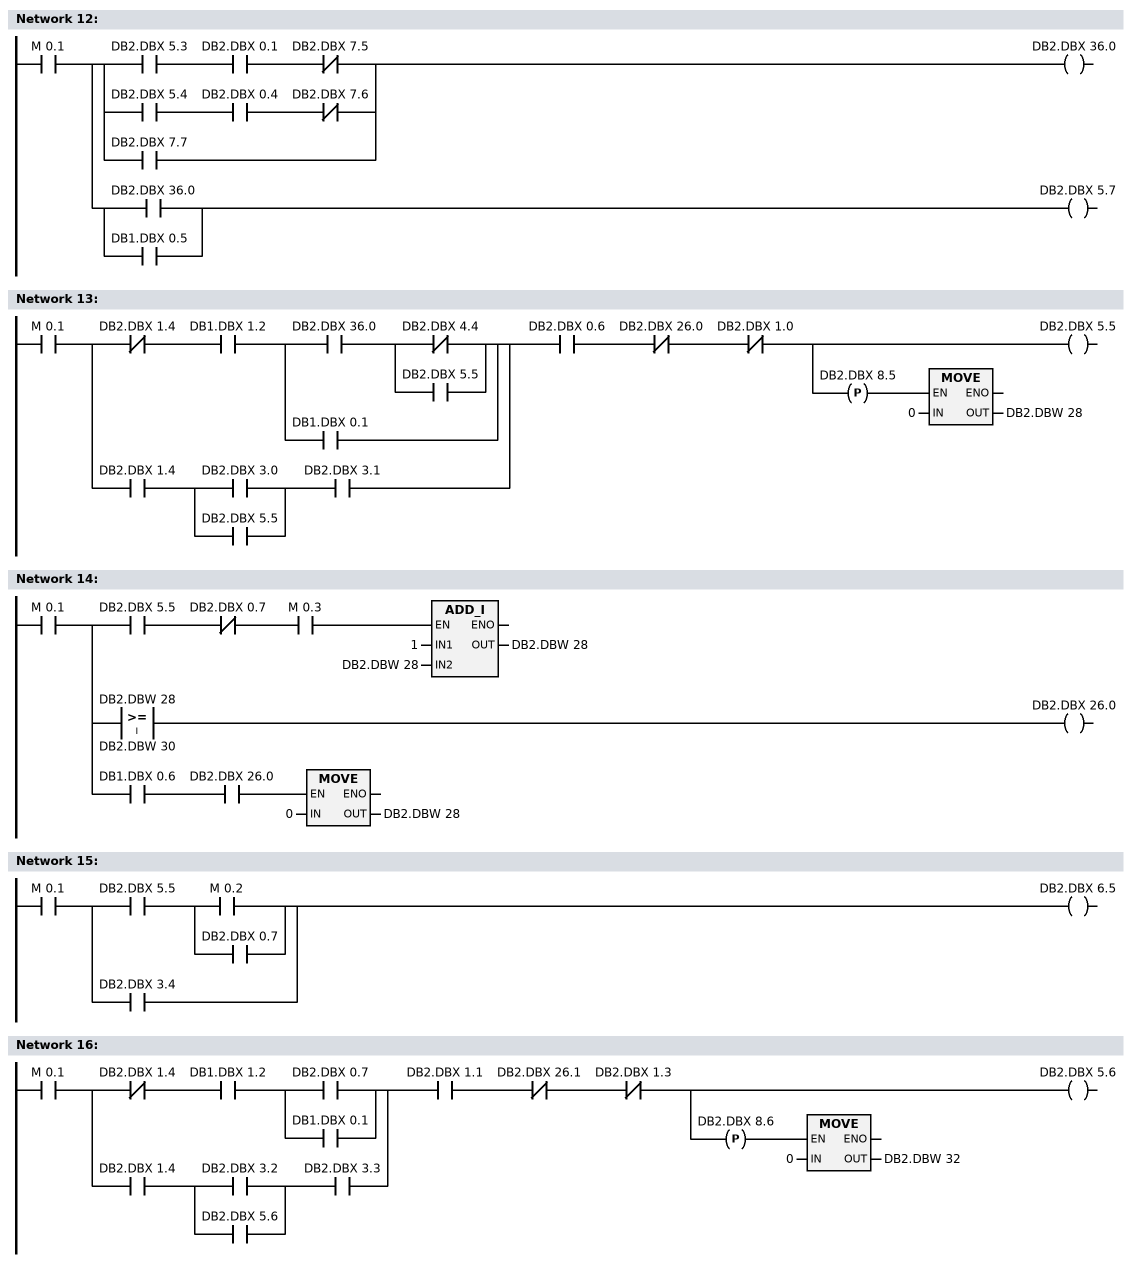
NETWORK
TITLE =
      A     M 0.1;
      =     L 0.0;
      A     L 0.0;
      A(;
      A     DB2.DBX 5.3;
      A     DB2.DBX 0.1;
      AN    DB2.DBX 7.5;
      O;
      A     DB2.DBX 5.4;
      A     DB2.DBX 0.4;
      AN    DB2.DBX 7.6;
      O     DB2.DBX 7.7;
      );
      =     DB2.DBX 36.0;
      A     L 0.0;
      A(;
      O     DB2.DBX 36.0;
      O     DB1.DBX 0.5;
      );
      =     DB2.DBX 5.7;
NETWORK
TITLE =
      A     M 0.1;
      A(;
      AN    DB2.DBX 1.4;
      A     DB1.DBX 1.2;
      A(;
      A     DB2.DBX 36.0;
      A(;
      ON    DB2.DBX 4.4;
      O     DB2.DBX 5.5;
      );
      O     DB1.DBX 0.1;
      );
      O;
      A     DB2.DBX 1.4;
      A(;
      O     DB2.DBX 3.0;
      O     DB2.DBX 5.5;
      );
      A     DB2.DBX 3.1;
      );
      A     DB2.DBX 0.6;
      AN    DB2.DBX 26.0;
      AN    DB2.DBX 1.0;
      =     L 0.0;
      A     L 0.0;
      BLD   102;
      =     DB2.DBX 5.5;
      A     L 0.0;
      FP    DB2.DBX 8.5;
      JNB   M011;
      L     0;
      T     DB2.DBW 28;
M011: NOP   0;
NETWORK
TITLE =
      A     M 0.1;
      =     L 0.0;
      A     L 0.0;
      A     DB2.DBX 5.5;
      AN    DB2.DBX 0.7;
      A     M 0.3;
      JNB   M012;
      L     1;
      L     DB2.DBW 28;
      +I;
      T     DB2.DBW 28;
M012: NOP   0;
      A     L 0.0;
      A(;
      L     DB2.DBW 28;
      L     DB2.DBW 30;
      >=I;
      );
      =     DB2.DBX 26.0;
      A     L 0.0;
      A     DB1.DBX 0.6;
      A     DB2.DBX 26.0;
      JNB   M013;
      L     0;
      T     DB2.DBW 28;
M013: NOP   0;
NETWORK
TITLE =
      A     M 0.1;
      A(;
      A     DB2.DBX 5.5;
      A(;
      O     M 0.2;
      O     DB2.DBX 0.7;
      );
      O     DB2.DBX 3.4;
      );
      =     DB2.DBX 6.5;
NETWORK
TITLE =
      A     M 0.1;
      A(;
      AN    DB2.DBX 1.4;
      A     DB1.DBX 1.2;
      A(;
      O     DB2.DBX 0.7;
      O     DB1.DBX 0.1;
      );
      O;
      A     DB2.DBX 1.4;
      A(;
      O     DB2.DBX 3.2;
      O     DB2.DBX 5.6;
      );
      A     DB2.DBX 3.3;
      );
      A     DB2.DBX 1.1;
      AN    DB2.DBX 26.1;
      AN    DB2.DBX 1.3;
      =     L 0.0;
      A     L 0.0;
      BLD   102;
      =     DB2.DBX 5.6;
      A     L 0.0;
      FP    DB2.DBX 8.6;
      JNB   M014;
      L     0;
      T     DB2.DBW 32;
M014: NOP   0;
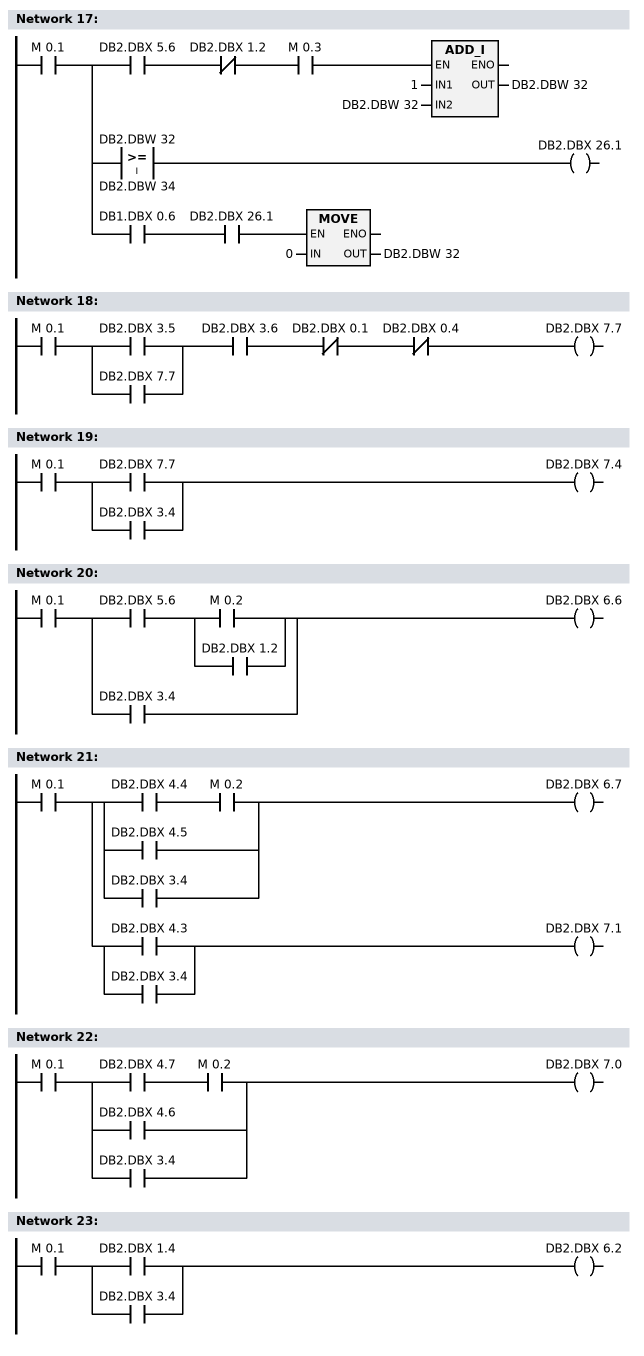
NETWORK
TITLE =
      A     M 0.1;
      =     L 0.0;
      A     L 0.0;
      A     DB2.DBX 5.6;
      AN    DB2.DBX 1.2;
      A     M 0.3;
      JNB   M015;
      L     1;
      L     DB2.DBW 32;
      +I;
      T     DB2.DBW 32;
M015: NOP   0;
      A     L 0.0;
      A(;
      L     DB2.DBW 32;
      L     DB2.DBW 34;
      >=I;
      );
      =     DB2.DBX 26.1;
      A     L 0.0;
      A     DB1.DBX 0.6;
      A     DB2.DBX 26.1;
      JNB   M016;
      L     0;
      T     DB2.DBW 32;
M016: NOP   0;
NETWORK
TITLE =
      A     M 0.1;
      A(;
      O     DB2.DBX 3.5;
      O     DB2.DBX 7.7;
      );
      A     DB2.DBX 3.6;
      AN    DB2.DBX 0.1;
      AN    DB2.DBX 0.4;
      =     DB2.DBX 7.7;
NETWORK
TITLE =
      A     M 0.1;
      A(;
      O     DB2.DBX 7.7;
      O     DB2.DBX 3.4;
      );
      =     DB2.DBX 7.4;
NETWORK
TITLE =
      A     M 0.1;
      A(;
      A     DB2.DBX 5.6;
      A(;
      O     M 0.2;
      O     DB2.DBX 1.2;
      );
      O     DB2.DBX 3.4;
      );
      =     DB2.DBX 6.6;
NETWORK
TITLE =
      A     M 0.1;
      =     L 0.0;
      A     L 0.0;
      A(;
      A     DB2.DBX 4.4;
      A     M 0.2;
      O     DB2.DBX 4.5;
      O     DB2.DBX 3.4;
      );
      =     DB2.DBX 6.7;
      A     L 0.0;
      A(;
      O     DB2.DBX 4.3;
      O     DB2.DBX 3.4;
      );
      =     DB2.DBX 7.1;
NETWORK
TITLE =
      A     M 0.1;
      A(;
      A     DB2.DBX 4.7;
      A     M 0.2;
      O     DB2.DBX 4.6;
      O     DB2.DBX 3.4;
      );
      =     DB2.DBX 7.0;
NETWORK
TITLE =
      A     M 0.1;
      A(;
      O     DB2.DBX 1.4;
      O     DB2.DBX 3.4;
      );
      =     DB2.DBX 6.2;
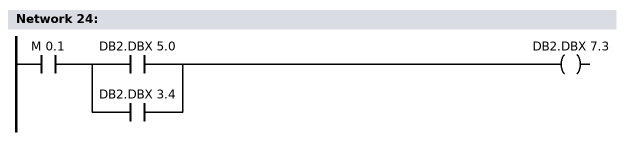
NETWORK
TITLE =
      A     M 0.1;
      A(;
      O     DB2.DBX 5.0;
      O     DB2.DBX 3.4;
      );
      =     DB2.DBX 7.3;
END_FUNCTION

FUNCTION FC 5 : VOID
AUTHOR : Kamillas
VERSION : 0.1
BEGIN
// (block stored without names or comments; labels and parameter names are numbered)
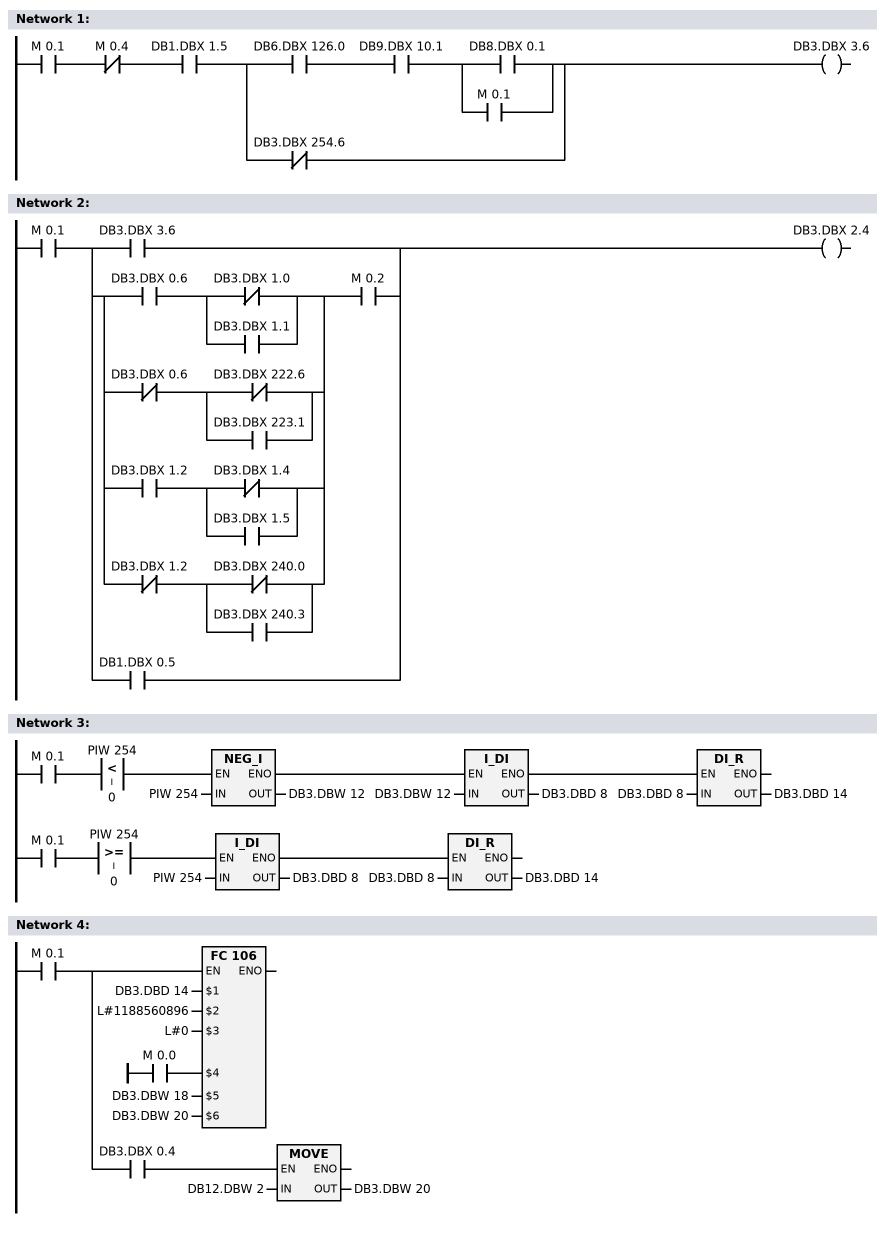
NETWORK
TITLE =
      A     M 0.1;
      AN    M 0.4;
      A     DB1.DBX 1.5;
      A(;
      A     DB6.DBX 126.0;
      A     DB9.DBX 10.1;
      A(;
      O     DB8.DBX 0.1;
      O     M 0.1;
      );
      ON    DB3.DBX 254.6;
      );
      =     DB3.DBX 3.6;
NETWORK
TITLE =
      A     M 0.1;
      A(;
      O     DB3.DBX 3.6;
      O;
      A(;
      A     DB3.DBX 0.6;
      A(;
      ON    DB3.DBX 1.0;
      O     DB3.DBX 1.1;
      );
      O;
      AN    DB3.DBX 0.6;
      A(;
      ON    DB3.DBX 222.6;
      O     DB3.DBX 223.1;
      );
      O;
      A     DB3.DBX 1.2;
      A(;
      ON    DB3.DBX 1.4;
      O     DB3.DBX 1.5;
      );
      O;
      AN    DB3.DBX 1.2;
      A(;
      ON    DB3.DBX 240.0;
      O     DB3.DBX 240.3;
      );
      );
      A     M 0.2;
      O     DB1.DBX 0.5;
      );
      =     DB3.DBX 2.4;
NETWORK
TITLE =
      A     M 0.1;
      =     L 0.0;
      A(;
      A(;
      A     L 0.0;
      A(;
      L     PIW 254;
      L     0;
      <I;
      );
      JNB   M001;
      L     PIW 254;
      NEGI;
      T     DB3.DBW 12;
      AN    OV;
      SAVE;
      CLR;
M001: A     BR;
      );
      JNB   M002;
      L     DB3.DBW 12;
      ITD;
      T     DB3.DBD 8;
      SET;
      SAVE;
      CLR;
M002: A     BR;
      );
      JNB   M003;
      L     DB3.DBD 8;
      DTR;
      T     DB3.DBD 14;
M003: NOP   0;
      A(;
      A     L 0.0;
      A(;
      L     PIW 254;
      L     0;
      >=I;
      );
      JNB   M004;
      L     PIW 254;
      ITD;
      T     DB3.DBD 8;
      SET;
      SAVE;
      CLR;
M004: A     BR;
      );
      JNB   M005;
      L     DB3.DBD 8;
      DTR;
      T     DB3.DBD 14;
M005: NOP   0;
NETWORK
TITLE =
      A     M 0.1;
      =     L 0.0;
      A     M 0.0;
      =     L 0.1;
      BLD   103;
      A     L 0.0;
      JNB   M006;
      CALL  FC 106 (
           $1                       := DB3.DBD 14,
           $2                       := L#1188560896,
           $3                       := L#0,
           $4                       := L 0.1,
           $5                       := DB3.DBW 18,
           $6                       := DB3.DBW 20);
M006: NOP   0;
      A     L 0.0;
      A     DB3.DBX 0.4;
      JNB   M007;
      L     DB12.DBW 2;
      T     DB3.DBW 20;
M007: NOP   0;
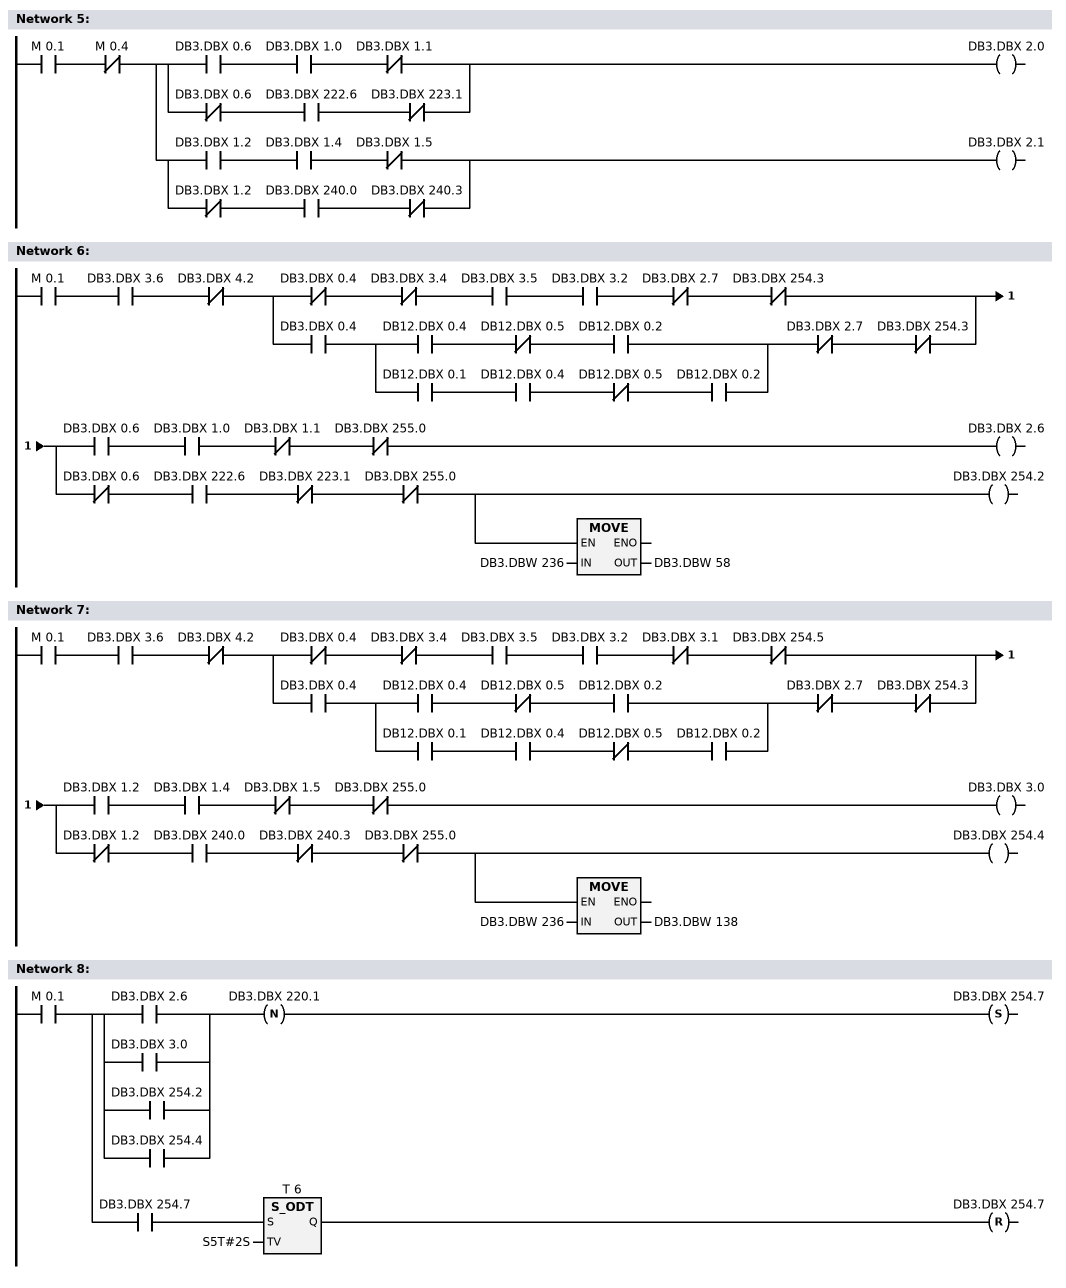
NETWORK
TITLE =
      A     M 0.1;
      AN    M 0.4;
      =     L 0.0;
      A     L 0.0;
      A(;
      A     DB3.DBX 0.6;
      A     DB3.DBX 1.0;
      AN    DB3.DBX 1.1;
      O;
      AN    DB3.DBX 0.6;
      A     DB3.DBX 222.6;
      AN    DB3.DBX 223.1;
      );
      =     DB3.DBX 2.0;
      A     L 0.0;
      A(;
      A     DB3.DBX 1.2;
      A     DB3.DBX 1.4;
      AN    DB3.DBX 1.5;
      O;
      AN    DB3.DBX 1.2;
      A     DB3.DBX 240.0;
      AN    DB3.DBX 240.3;
      );
      =     DB3.DBX 2.1;
NETWORK
TITLE =
      A     M 0.1;
      A     DB3.DBX 3.6;
      AN    DB3.DBX 4.2;
      A(;
      AN    DB3.DBX 0.4;
      AN    DB3.DBX 3.4;
      A     DB3.DBX 3.5;
      A     DB3.DBX 3.2;
      AN    DB3.DBX 2.7;
      AN    DB3.DBX 254.3;
      O;
      A     DB3.DBX 0.4;
      A(;
      A     DB12.DBX 0.4;
      AN    DB12.DBX 0.5;
      A     DB12.DBX 0.2;
      O;
      A     DB12.DBX 0.1;
      A     DB12.DBX 0.4;
      AN    DB12.DBX 0.5;
      A     DB12.DBX 0.2;
      );
      AN    DB3.DBX 2.7;
      AN    DB3.DBX 254.3;
      );
      =     L 0.0;
      A     L 0.0;
      A     DB3.DBX 0.6;
      A     DB3.DBX 1.0;
      AN    DB3.DBX 1.1;
      AN    DB3.DBX 255.0;
      =     DB3.DBX 2.6;
      A     L 0.0;
      AN    DB3.DBX 0.6;
      A     DB3.DBX 222.6;
      AN    DB3.DBX 223.1;
      AN    DB3.DBX 255.0;
      =     L 0.1;
      A     L 0.1;
      BLD   102;
      =     DB3.DBX 254.2;
      A     L 0.1;
      JNB   M008;
      L     DB3.DBW 236;
      T     DB3.DBW 58;
M008: NOP   0;
NETWORK
TITLE =
      A     M 0.1;
      A     DB3.DBX 3.6;
      AN    DB3.DBX 4.2;
      A(;
      AN    DB3.DBX 0.4;
      AN    DB3.DBX 3.4;
      A     DB3.DBX 3.5;
      A     DB3.DBX 3.2;
      AN    DB3.DBX 3.1;
      AN    DB3.DBX 254.5;
      O;
      A     DB3.DBX 0.4;
      A(;
      A     DB12.DBX 0.4;
      AN    DB12.DBX 0.5;
      A     DB12.DBX 0.2;
      O;
      A     DB12.DBX 0.1;
      A     DB12.DBX 0.4;
      AN    DB12.DBX 0.5;
      A     DB12.DBX 0.2;
      );
      AN    DB3.DBX 2.7;
      AN    DB3.DBX 254.3;
      );
      =     L 0.0;
      A     L 0.0;
      A     DB3.DBX 1.2;
      A     DB3.DBX 1.4;
      AN    DB3.DBX 1.5;
      AN    DB3.DBX 255.0;
      =     DB3.DBX 3.0;
      A     L 0.0;
      AN    DB3.DBX 1.2;
      A     DB3.DBX 240.0;
      AN    DB3.DBX 240.3;
      AN    DB3.DBX 255.0;
      =     L 0.1;
      A     L 0.1;
      BLD   102;
      =     DB3.DBX 254.4;
      A     L 0.1;
      JNB   M009;
      L     DB3.DBW 236;
      T     DB3.DBW 138;
M009: NOP   0;
NETWORK
TITLE =
      A     M 0.1;
      =     L 0.0;
      A     L 0.0;
      A(;
      O     DB3.DBX 2.6;
      O     DB3.DBX 3.0;
      O     DB3.DBX 254.2;
      O     DB3.DBX 254.4;
      );
      FN    DB3.DBX 220.1;
      S     DB3.DBX 254.7;
      A     L 0.0;
      A     DB3.DBX 254.7;
      L     S5T#2S;
      SD    T 6;
      NOP   0;
      NOP   0;
      NOP   0;
      A     T 6;
      R     DB3.DBX 254.7;
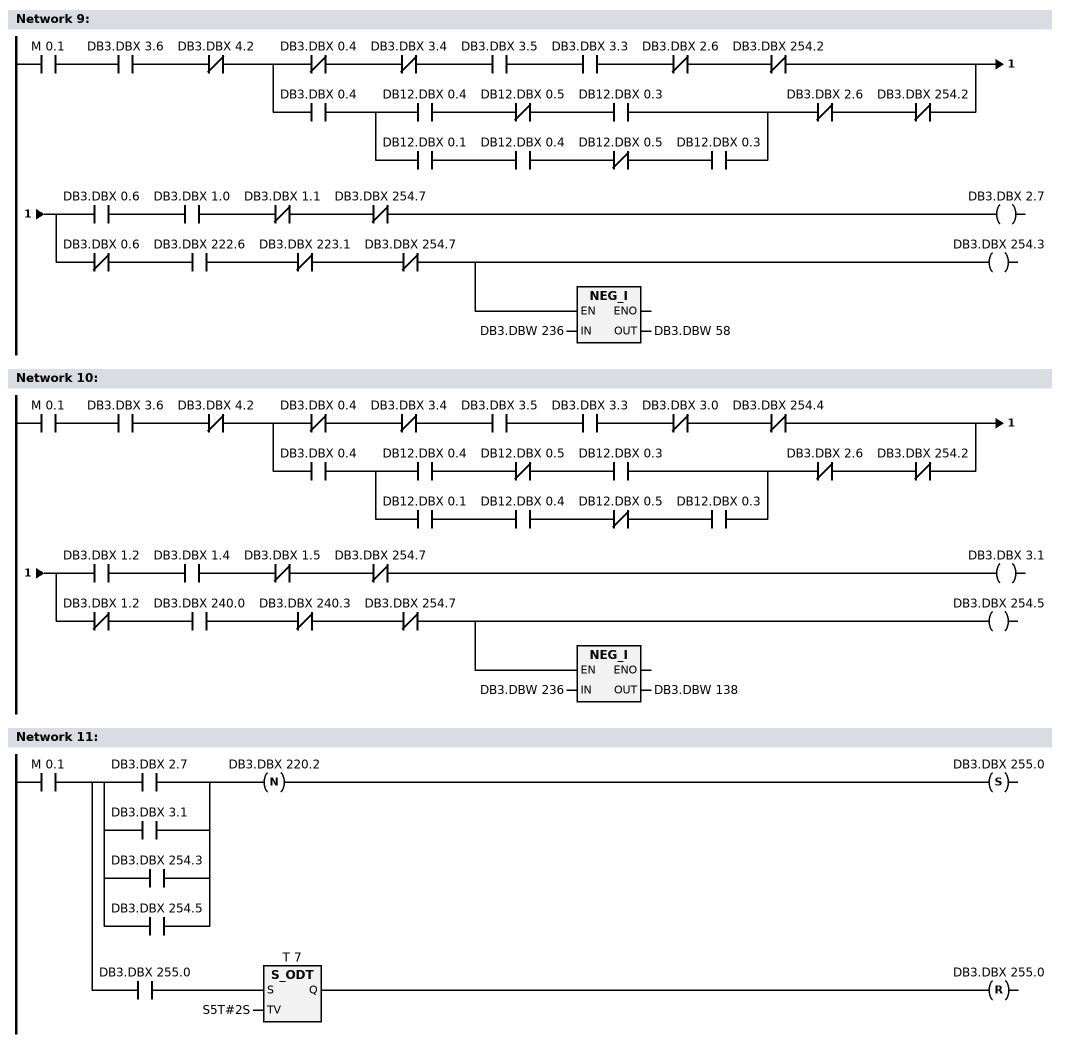
NETWORK
TITLE =
      A     M 0.1;
      A     DB3.DBX 3.6;
      AN    DB3.DBX 4.2;
      A(;
      AN    DB3.DBX 0.4;
      AN    DB3.DBX 3.4;
      A     DB3.DBX 3.5;
      A     DB3.DBX 3.3;
      AN    DB3.DBX 2.6;
      AN    DB3.DBX 254.2;
      O;
      A     DB3.DBX 0.4;
      A(;
      A     DB12.DBX 0.4;
      AN    DB12.DBX 0.5;
      A     DB12.DBX 0.3;
      O;
      A     DB12.DBX 0.1;
      A     DB12.DBX 0.4;
      AN    DB12.DBX 0.5;
      A     DB12.DBX 0.3;
      );
      AN    DB3.DBX 2.6;
      AN    DB3.DBX 254.2;
      );
      =     L 0.0;
      A     L 0.0;
      A     DB3.DBX 0.6;
      A     DB3.DBX 1.0;
      AN    DB3.DBX 1.1;
      AN    DB3.DBX 254.7;
      =     DB3.DBX 2.7;
      A     L 0.0;
      AN    DB3.DBX 0.6;
      A     DB3.DBX 222.6;
      AN    DB3.DBX 223.1;
      AN    DB3.DBX 254.7;
      =     L 0.1;
      A     L 0.1;
      BLD   102;
      =     DB3.DBX 254.3;
      A     L 0.1;
      JNB   M010;
      L     DB3.DBW 236;
      NEGI;
      T     DB3.DBW 58;
M010: NOP   0;
NETWORK
TITLE =
      A     M 0.1;
      A     DB3.DBX 3.6;
      AN    DB3.DBX 4.2;
      A(;
      AN    DB3.DBX 0.4;
      AN    DB3.DBX 3.4;
      A     DB3.DBX 3.5;
      A     DB3.DBX 3.3;
      AN    DB3.DBX 3.0;
      AN    DB3.DBX 254.4;
      O;
      A     DB3.DBX 0.4;
      A(;
      A     DB12.DBX 0.4;
      AN    DB12.DBX 0.5;
      A     DB12.DBX 0.3;
      O;
      A     DB12.DBX 0.1;
      A     DB12.DBX 0.4;
      AN    DB12.DBX 0.5;
      A     DB12.DBX 0.3;
      );
      AN    DB3.DBX 2.6;
      AN    DB3.DBX 254.2;
      );
      =     L 0.0;
      A     L 0.0;
      A     DB3.DBX 1.2;
      A     DB3.DBX 1.4;
      AN    DB3.DBX 1.5;
      AN    DB3.DBX 254.7;
      =     DB3.DBX 3.1;
      A     L 0.0;
      AN    DB3.DBX 1.2;
      A     DB3.DBX 240.0;
      AN    DB3.DBX 240.3;
      AN    DB3.DBX 254.7;
      =     L 0.1;
      A     L 0.1;
      BLD   102;
      =     DB3.DBX 254.5;
      A     L 0.1;
      JNB   M011;
      L     DB3.DBW 236;
      NEGI;
      T     DB3.DBW 138;
M011: NOP   0;
NETWORK
TITLE =
      A     M 0.1;
      =     L 0.0;
      A     L 0.0;
      A(;
      O     DB3.DBX 2.7;
      O     DB3.DBX 3.1;
      O     DB3.DBX 254.3;
      O     DB3.DBX 254.5;
      );
      FN    DB3.DBX 220.2;
      S     DB3.DBX 255.0;
      A     L 0.0;
      A     DB3.DBX 255.0;
      L     S5T#2S;
      SD    T 7;
      NOP   0;
      NOP   0;
      NOP   0;
      A     T 7;
      R     DB3.DBX 255.0;
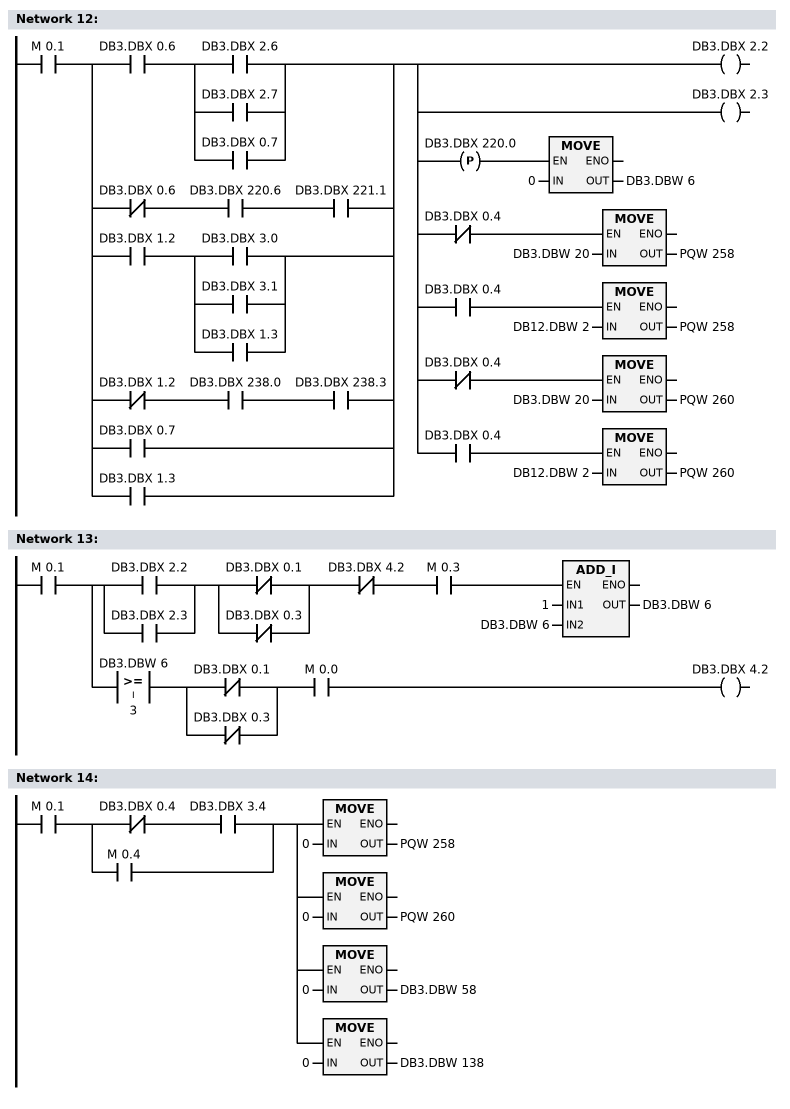
NETWORK
TITLE =
      A     M 0.1;
      A(;
      A     DB3.DBX 0.6;
      A(;
      O     DB3.DBX 2.6;
      O     DB3.DBX 2.7;
      O     DB3.DBX 0.7;
      );
      O;
      AN    DB3.DBX 0.6;
      A     DB3.DBX 220.6;
      A     DB3.DBX 221.1;
      O;
      A     DB3.DBX 1.2;
      A(;
      O     DB3.DBX 3.0;
      O     DB3.DBX 3.1;
      O     DB3.DBX 1.3;
      );
      O;
      AN    DB3.DBX 1.2;
      A     DB3.DBX 238.0;
      A     DB3.DBX 238.3;
      O     DB3.DBX 0.7;
      O     DB3.DBX 1.3;
      );
      =     L 0.0;
      A     L 0.0;
      BLD   102;
      =     DB3.DBX 2.2;
      A     L 0.0;
      BLD   102;
      =     DB3.DBX 2.3;
      A     L 0.0;
      FP    DB3.DBX 220.0;
      JNB   M012;
      L     0;
      T     DB3.DBW 6;
M012: NOP   0;
      A     L 0.0;
      AN    DB3.DBX 0.4;
      JNB   M013;
      L     DB3.DBW 20;
      T     PQW 258;
M013: NOP   0;
      A     L 0.0;
      A     DB3.DBX 0.4;
      JNB   M014;
      L     DB12.DBW 2;
      T     PQW 258;
M014: NOP   0;
      A     L 0.0;
      AN    DB3.DBX 0.4;
      JNB   M015;
      L     DB3.DBW 20;
      T     PQW 260;
M015: NOP   0;
      A     L 0.0;
      A     DB3.DBX 0.4;
      JNB   M016;
      L     DB12.DBW 2;
      T     PQW 260;
M016: NOP   0;
NETWORK
TITLE =
      A     M 0.1;
      =     L 0.0;
      A     L 0.0;
      A(;
      O     DB3.DBX 2.2;
      O     DB3.DBX 2.3;
      );
      A(;
      ON    DB3.DBX 0.1;
      ON    DB3.DBX 0.3;
      );
      AN    DB3.DBX 4.2;
      A     M 0.3;
      JNB   M017;
      L     1;
      L     DB3.DBW 6;
      +I;
      T     DB3.DBW 6;
M017: NOP   0;
      A     L 0.0;
      A(;
      L     DB3.DBW 6;
      L     3;
      >=I;
      );
      A(;
      ON    DB3.DBX 0.1;
      ON    DB3.DBX 0.3;
      );
      A     M 0.0;
      =     DB3.DBX 4.2;
NETWORK
TITLE =
      A     M 0.1;
      A(;
      AN    DB3.DBX 0.4;
      A     DB3.DBX 3.4;
      O     M 0.4;
      );
      =     L 0.0;
      A     L 0.0;
      JNB   M018;
      L     0;
      T     PQW 258;
M018: NOP   0;
      A     L 0.0;
      JNB   M019;
      L     0;
      T     PQW 260;
M019: NOP   0;
      A     L 0.0;
      JNB   M020;
      L     0;
      T     DB3.DBW 58;
M020: NOP   0;
      A     L 0.0;
      JNB   M021;
      L     0;
      T     DB3.DBW 138;
M021: NOP   0;
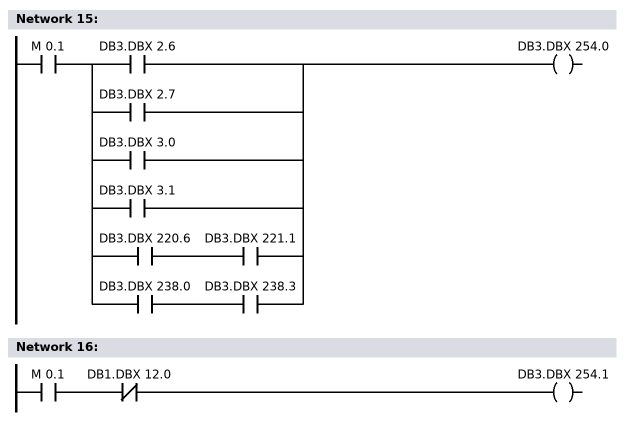
NETWORK
TITLE =
      A     M 0.1;
      A(;
      O     DB3.DBX 2.6;
      O     DB3.DBX 2.7;
      O     DB3.DBX 3.0;
      O     DB3.DBX 3.1;
      O;
      A     DB3.DBX 220.6;
      A     DB3.DBX 221.1;
      O;
      A     DB3.DBX 238.0;
      A     DB3.DBX 238.3;
      );
      =     DB3.DBX 254.0;
NETWORK
TITLE =
      A     M 0.1;
      AN    DB1.DBX 12.0;
      =     DB3.DBX 254.1;
END_FUNCTION

FUNCTION FC 6 : VOID
AUTHOR : Kamillas
VERSION : 0.1
BEGIN
// (block stored without names or comments; labels and parameter names are numbered)
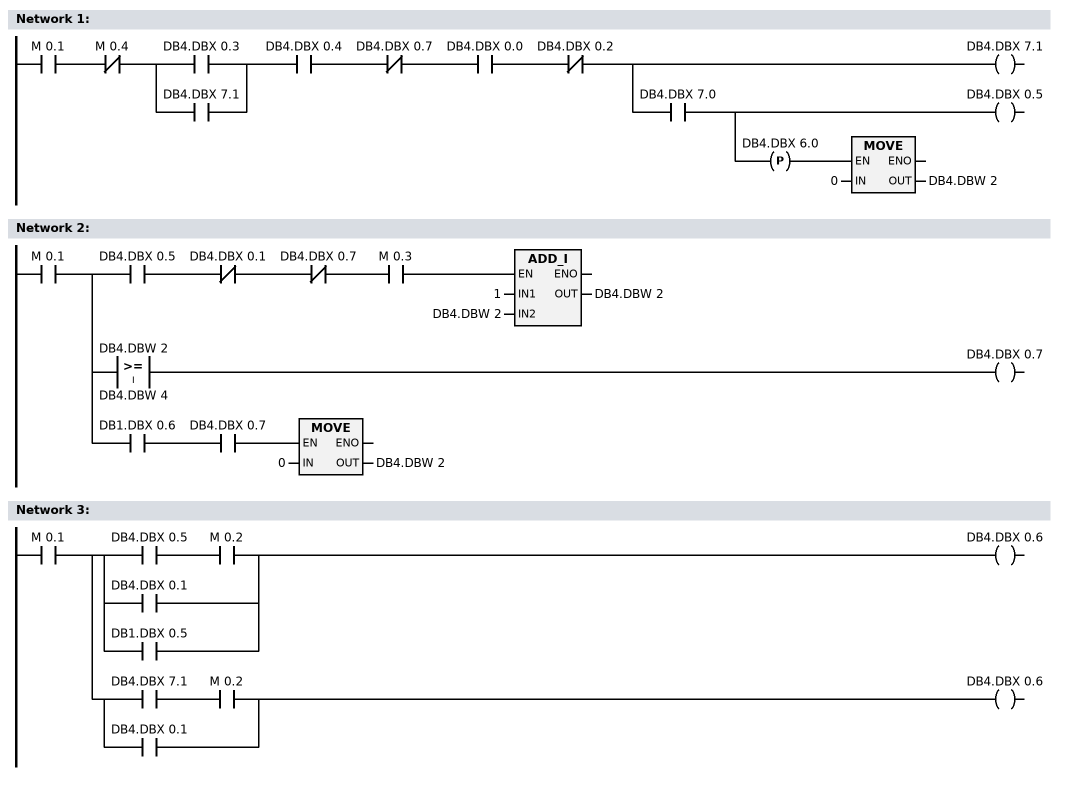
NETWORK
TITLE =
      A     M 0.1;
      AN    M 0.4;
      A(;
      O     DB4.DBX 0.3;
      O     DB4.DBX 7.1;
      );
      A     DB4.DBX 0.4;
      AN    DB4.DBX 0.7;
      A     DB4.DBX 0.0;
      AN    DB4.DBX 0.2;
      =     L 0.0;
      A     L 0.0;
      BLD   102;
      =     DB4.DBX 7.1;
      A     L 0.0;
      A     DB4.DBX 7.0;
      =     L 0.1;
      A     L 0.1;
      BLD   102;
      =     DB4.DBX 0.5;
      A     L 0.1;
      FP    DB4.DBX 6.0;
      JNB   M001;
      L     0;
      T     DB4.DBW 2;
M001: NOP   0;
NETWORK
TITLE =
      A     M 0.1;
      =     L 0.0;
      A     L 0.0;
      A     DB4.DBX 0.5;
      AN    DB4.DBX 0.1;
      AN    DB4.DBX 0.7;
      A     M 0.3;
      JNB   M002;
      L     1;
      L     DB4.DBW 2;
      +I;
      T     DB4.DBW 2;
M002: NOP   0;
      A     L 0.0;
      A(;
      L     DB4.DBW 2;
      L     DB4.DBW 4;
      >=I;
      );
      =     DB4.DBX 0.7;
      A     L 0.0;
      A     DB1.DBX 0.6;
      A     DB4.DBX 0.7;
      JNB   M003;
      L     0;
      T     DB4.DBW 2;
M003: NOP   0;
NETWORK
TITLE =
      A     M 0.1;
      =     L 0.0;
      A     L 0.0;
      A(;
      A     DB4.DBX 0.5;
      A     M 0.2;
      O     DB4.DBX 0.1;
      O     DB1.DBX 0.5;
      );
      =     DB4.DBX 0.6;
      A     L 0.0;
      A(;
      A     DB4.DBX 7.1;
      A     M 0.2;
      O     DB4.DBX 0.1;
      );
      =     DB4.DBX 0.6;
END_FUNCTION

FUNCTION FC 7 : VOID
AUTHOR : Kamillas
VERSION : 0.1
BEGIN
// (block stored without names or comments; labels and parameter names are numbered)
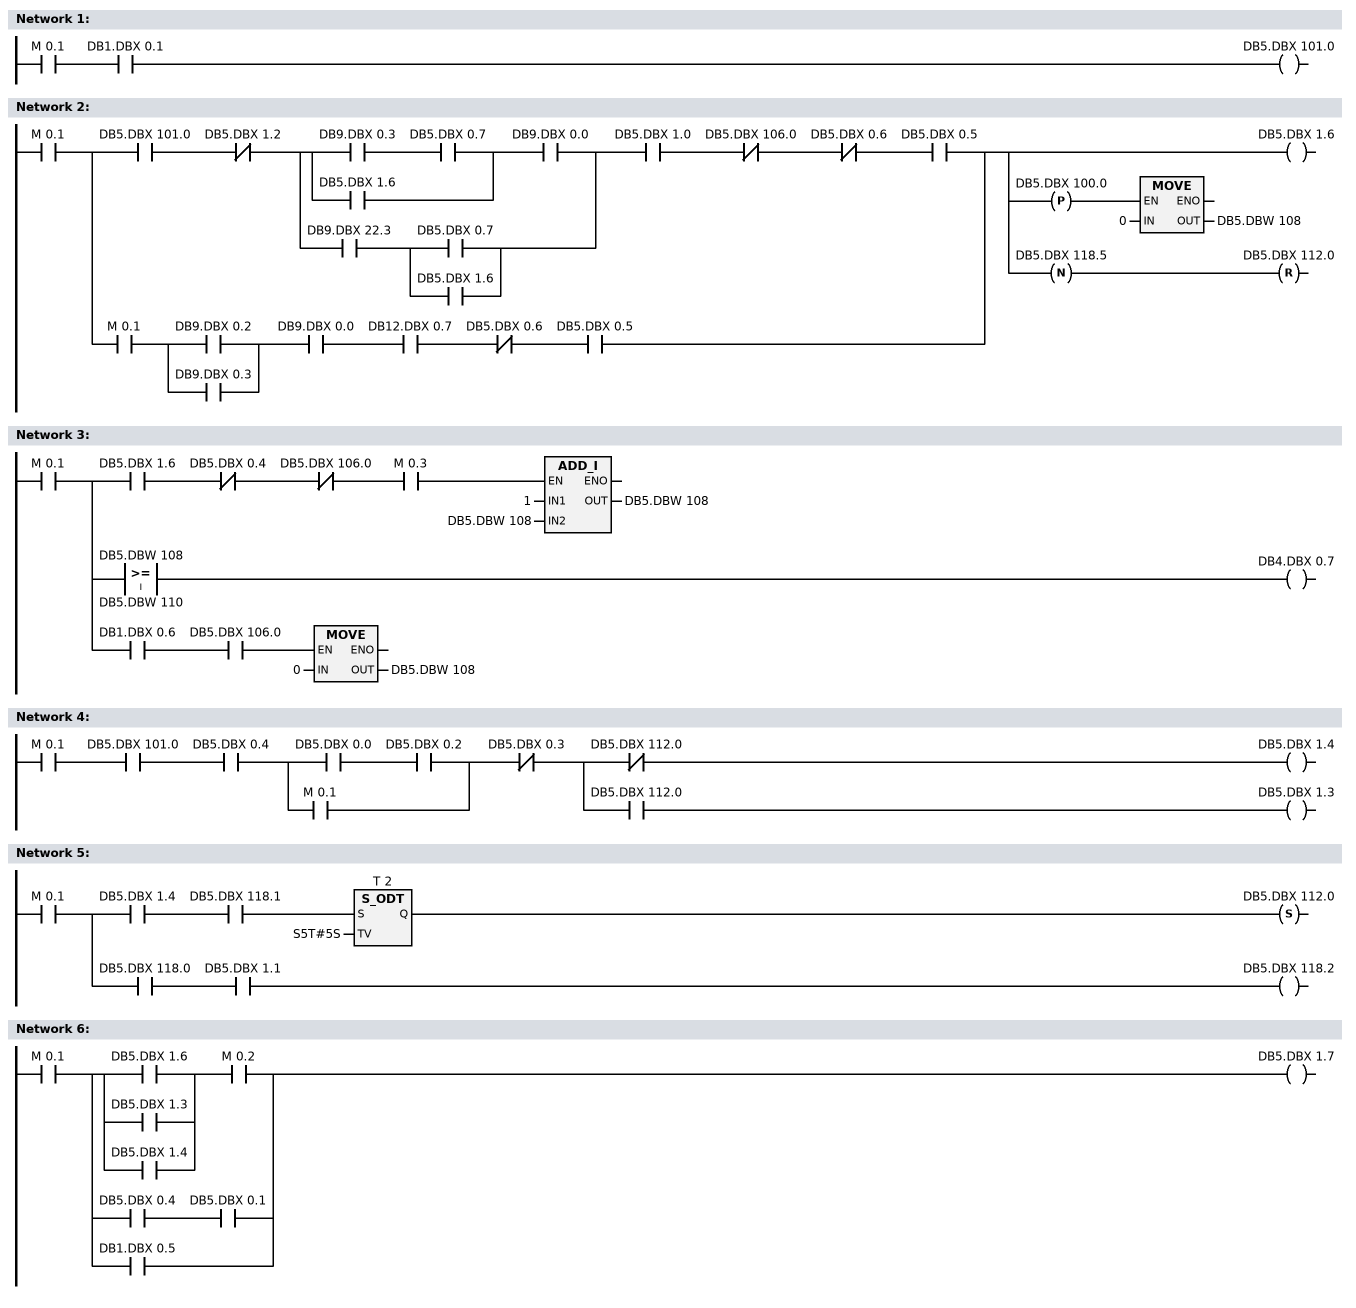
NETWORK
TITLE =
      A     M 0.1;
      A     DB1.DBX 0.1;
      =     DB5.DBX 101.0;
NETWORK
TITLE =
      A     M 0.1;
      A(;
      A     DB5.DBX 101.0;
      AN    DB5.DBX 1.2;
      A(;
      A(;
      A     DB9.DBX 0.3;
      A     DB5.DBX 0.7;
      O     DB5.DBX 1.6;
      );
      A     DB9.DBX 0.0;
      O;
      A     DB9.DBX 22.3;
      A(;
      O     DB5.DBX 0.7;
      O     DB5.DBX 1.6;
      );
      );
      A     DB5.DBX 1.0;
      AN    DB5.DBX 106.0;
      AN    DB5.DBX 0.6;
      A     DB5.DBX 0.5;
      O;
      A     M 0.1;
      A(;
      O     DB9.DBX 0.2;
      O     DB9.DBX 0.3;
      );
      A     DB9.DBX 0.0;
      A     DB12.DBX 0.7;
      AN    DB5.DBX 0.6;
      A     DB5.DBX 0.5;
      );
      =     L 0.0;
      A     L 0.0;
      BLD   102;
      =     DB5.DBX 1.6;
      A     L 0.0;
      FP    DB5.DBX 100.0;
      JNB   M001;
      L     0;
      T     DB5.DBW 108;
M001: NOP   0;
      A     L 0.0;
      FN    DB5.DBX 118.5;
      R     DB5.DBX 112.0;
NETWORK
TITLE =
      A     M 0.1;
      =     L 0.0;
      A     L 0.0;
      A     DB5.DBX 1.6;
      AN    DB5.DBX 0.4;
      AN    DB5.DBX 106.0;
      A     M 0.3;
      JNB   M002;
      L     1;
      L     DB5.DBW 108;
      +I;
      T     DB5.DBW 108;
M002: NOP   0;
      A     L 0.0;
      A(;
      L     DB5.DBW 108;
      L     DB5.DBW 110;
      >=I;
      );
      =     DB4.DBX 0.7;
      A     L 0.0;
      A     DB1.DBX 0.6;
      A     DB5.DBX 106.0;
      JNB   M003;
      L     0;
      T     DB5.DBW 108;
M003: NOP   0;
NETWORK
TITLE =
      A     M 0.1;
      A     DB5.DBX 101.0;
      A     DB5.DBX 0.4;
      A(;
      A     DB5.DBX 0.0;
      A     DB5.DBX 0.2;
      O     M 0.1;
      );
      AN    DB5.DBX 0.3;
      =     L 0.0;
      A     L 0.0;
      AN    DB5.DBX 112.0;
      =     DB5.DBX 1.4;
      A     L 0.0;
      A     DB5.DBX 112.0;
      =     DB5.DBX 1.3;
NETWORK
TITLE =
      A     M 0.1;
      =     L 0.0;
      A     L 0.0;
      A     DB5.DBX 1.4;
      A     DB5.DBX 118.1;
      L     S5T#5S;
      SD    T 2;
      NOP   0;
      NOP   0;
      NOP   0;
      A     T 2;
      S     DB5.DBX 112.0;
      A     L 0.0;
      A     DB5.DBX 118.0;
      A     DB5.DBX 1.1;
      =     DB5.DBX 118.2;
NETWORK
TITLE =
      A     M 0.1;
      A(;
      A(;
      O     DB5.DBX 1.6;
      O     DB5.DBX 1.3;
      O     DB5.DBX 1.4;
      );
      A     M 0.2;
      O;
      A     DB5.DBX 0.4;
      A     DB5.DBX 0.1;
      O     DB1.DBX 0.5;
      );
      =     DB5.DBX 1.7;
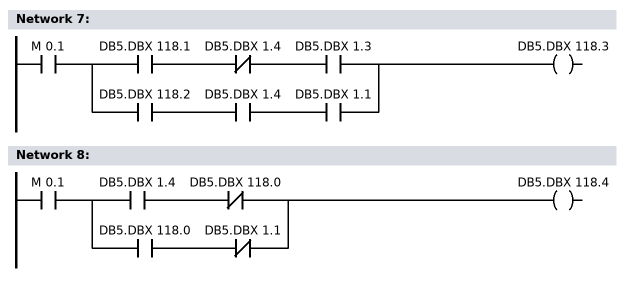
NETWORK
TITLE =
      A     M 0.1;
      A(;
      A     DB5.DBX 118.1;
      AN    DB5.DBX 1.4;
      A     DB5.DBX 1.3;
      O;
      A     DB5.DBX 118.2;
      A     DB5.DBX 1.4;
      A     DB5.DBX 1.1;
      );
      =     DB5.DBX 118.3;
NETWORK
TITLE =
      A     M 0.1;
      A(;
      A     DB5.DBX 1.4;
      AN    DB5.DBX 118.0;
      O;
      A     DB5.DBX 118.0;
      AN    DB5.DBX 1.1;
      );
      =     DB5.DBX 118.4;
END_FUNCTION

FUNCTION FC 8 : VOID
AUTHOR : Kamillas
VERSION : 0.1
BEGIN
// (block stored without names or comments; labels and parameter names are numbered)
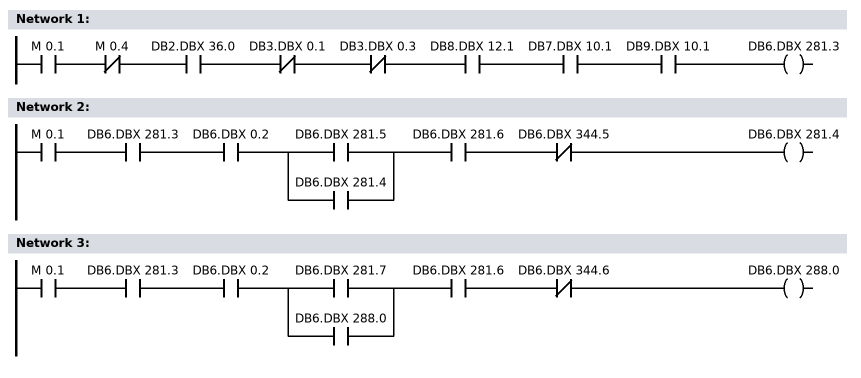
NETWORK
TITLE =
      A     M 0.1;
      AN    M 0.4;
      A     DB2.DBX 36.0;
      AN    DB3.DBX 0.1;
      AN    DB3.DBX 0.3;
      A     DB8.DBX 12.1;
      A     DB7.DBX 10.1;
      A     DB9.DBX 10.1;
      =     DB6.DBX 281.3;
NETWORK
TITLE =
      A     M 0.1;
      A     DB6.DBX 281.3;
      A     DB6.DBX 0.2;
      A(;
      O     DB6.DBX 281.5;
      O     DB6.DBX 281.4;
      );
      A     DB6.DBX 281.6;
      AN    DB6.DBX 344.5;
      =     DB6.DBX 281.4;
NETWORK
TITLE =
      A     M 0.1;
      A     DB6.DBX 281.3;
      A     DB6.DBX 0.2;
      A(;
      O     DB6.DBX 281.7;
      O     DB6.DBX 288.0;
      );
      A     DB6.DBX 281.6;
      AN    DB6.DBX 344.6;
      =     DB6.DBX 288.0;
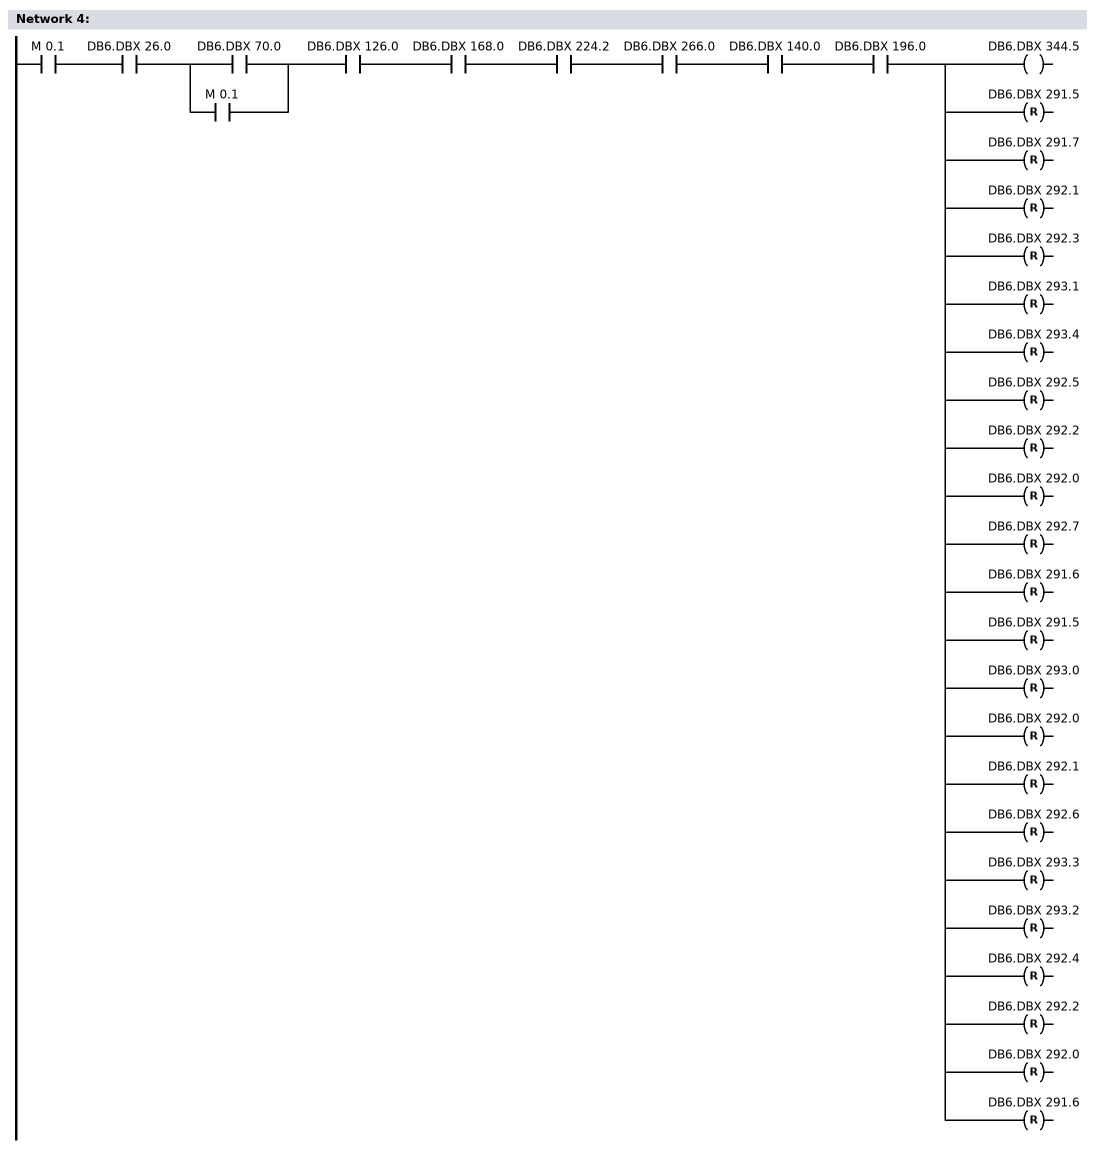
NETWORK
TITLE =
      A     M 0.1;
      A     DB6.DBX 26.0;
      A(;
      O     DB6.DBX 70.0;
      O     M 0.1;
      );
      A     DB6.DBX 126.0;
      A     DB6.DBX 168.0;
      A     DB6.DBX 224.2;
      A     DB6.DBX 266.0;
      A     DB6.DBX 140.0;
      A     DB6.DBX 196.0;
      =     DB6.DBX 344.5;
      R     DB6.DBX 291.5;
      R     DB6.DBX 291.7;
      R     DB6.DBX 292.1;
      R     DB6.DBX 292.3;
      R     DB6.DBX 293.1;
      R     DB6.DBX 293.4;
      R     DB6.DBX 292.5;
      R     DB6.DBX 292.2;
      R     DB6.DBX 292.0;
      R     DB6.DBX 292.7;
      R     DB6.DBX 291.6;
      R     DB6.DBX 291.5;
      R     DB6.DBX 293.0;
      R     DB6.DBX 292.0;
      R     DB6.DBX 292.1;
      R     DB6.DBX 292.6;
      R     DB6.DBX 293.3;
      R     DB6.DBX 293.2;
      R     DB6.DBX 292.4;
      R     DB6.DBX 292.2;
      R     DB6.DBX 292.0;
      R     DB6.DBX 291.6;
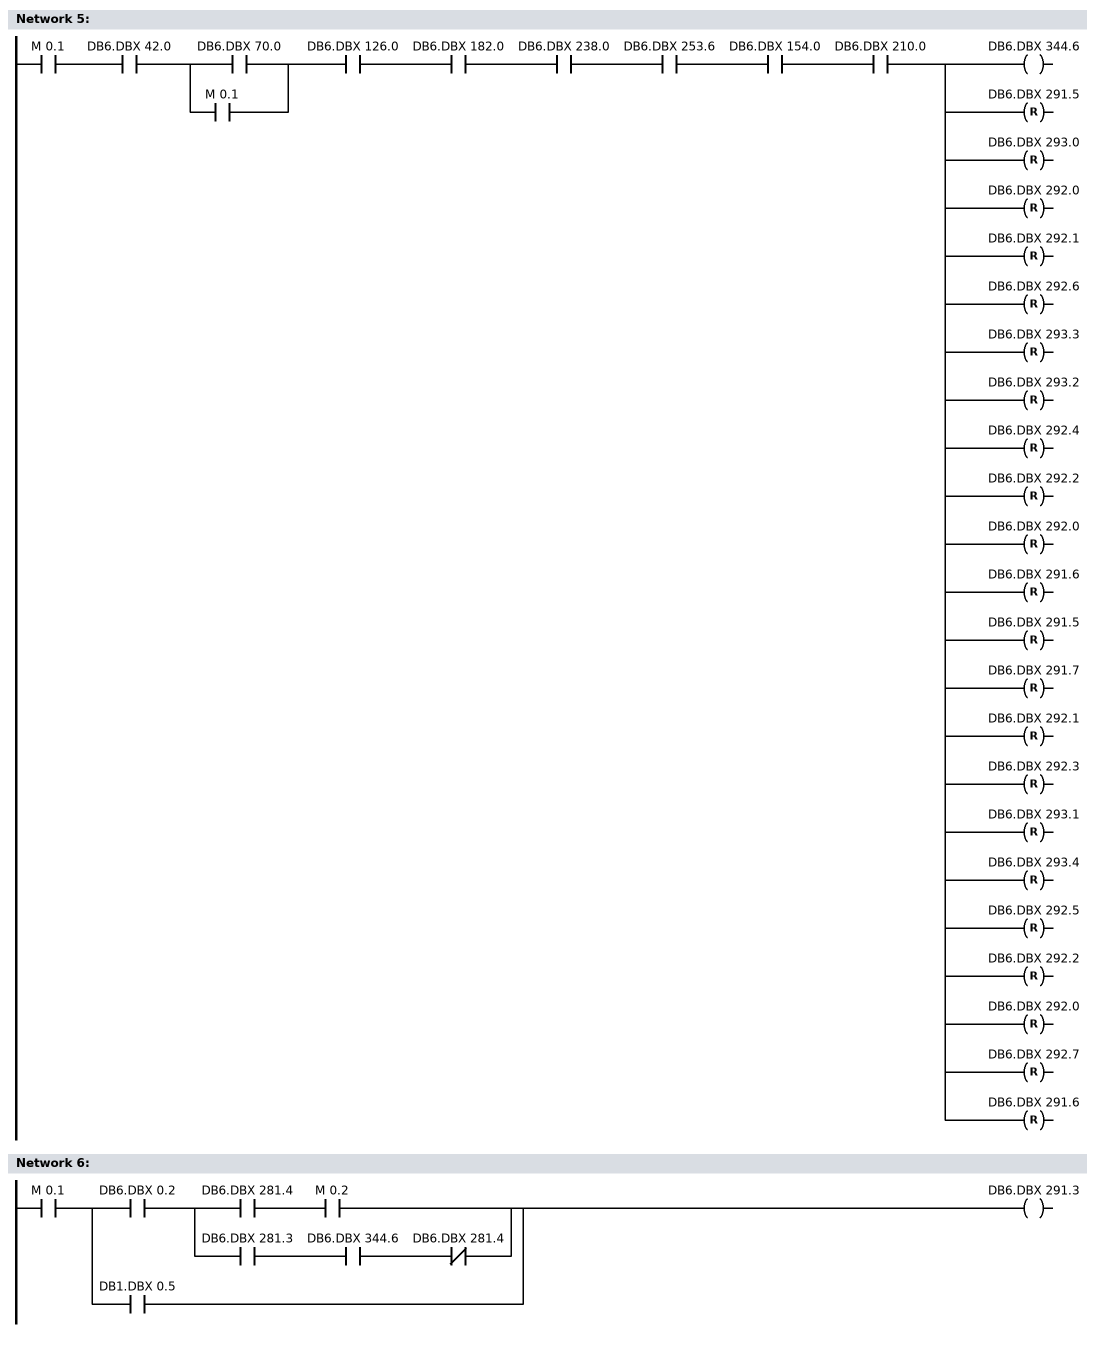
NETWORK
TITLE =
      A     M 0.1;
      A     DB6.DBX 42.0;
      A(;
      O     DB6.DBX 70.0;
      O     M 0.1;
      );
      A     DB6.DBX 126.0;
      A     DB6.DBX 182.0;
      A     DB6.DBX 238.0;
      A     DB6.DBX 253.6;
      A     DB6.DBX 154.0;
      A     DB6.DBX 210.0;
      =     DB6.DBX 344.6;
      R     DB6.DBX 291.5;
      R     DB6.DBX 293.0;
      R     DB6.DBX 292.0;
      R     DB6.DBX 292.1;
      R     DB6.DBX 292.6;
      R     DB6.DBX 293.3;
      R     DB6.DBX 293.2;
      R     DB6.DBX 292.4;
      R     DB6.DBX 292.2;
      R     DB6.DBX 292.0;
      R     DB6.DBX 291.6;
      R     DB6.DBX 291.5;
      R     DB6.DBX 291.7;
      R     DB6.DBX 292.1;
      R     DB6.DBX 292.3;
      R     DB6.DBX 293.1;
      R     DB6.DBX 293.4;
      R     DB6.DBX 292.5;
      R     DB6.DBX 292.2;
      R     DB6.DBX 292.0;
      R     DB6.DBX 292.7;
      R     DB6.DBX 291.6;
NETWORK
TITLE =
      A     M 0.1;
      A(;
      A     DB6.DBX 0.2;
      A(;
      A     DB6.DBX 281.4;
      A     M 0.2;
      O;
      A     DB6.DBX 281.3;
      A     DB6.DBX 344.6;
      AN    DB6.DBX 281.4;
      );
      O     DB1.DBX 0.5;
      );
      =     DB6.DBX 291.3;
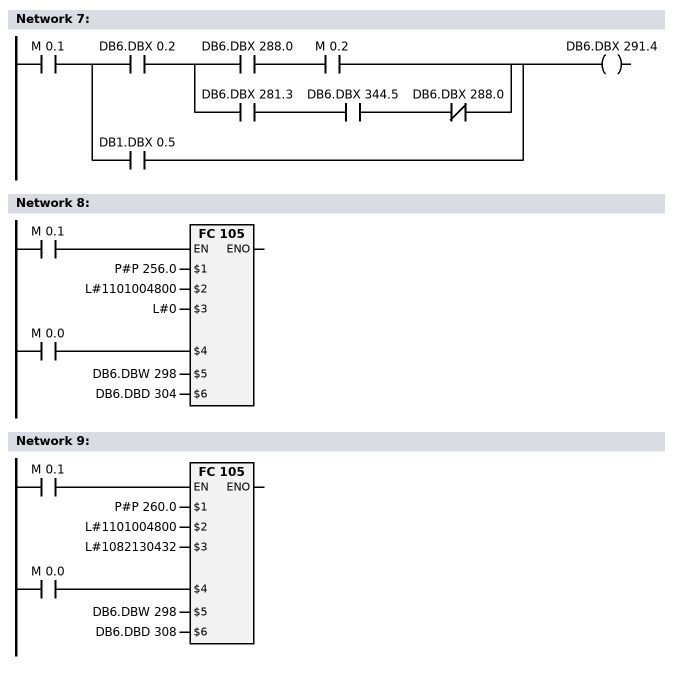
NETWORK
TITLE =
      A     M 0.1;
      A(;
      A     DB6.DBX 0.2;
      A(;
      A     DB6.DBX 288.0;
      A     M 0.2;
      O;
      A     DB6.DBX 281.3;
      A     DB6.DBX 344.5;
      AN    DB6.DBX 288.0;
      );
      O     DB1.DBX 0.5;
      );
      =     DB6.DBX 291.4;
NETWORK
TITLE =
      A     M 0.0;
      =     L 0.0;
      BLD   103;
      A     M 0.1;
      JNB   M001;
      CALL  FC 105 (
           $1                       := P#P 256.0,
           $2                       := L#1101004800,
           $3                       := L#0,
           $4                       := L 0.0,
           $5                       := DB6.DBW 298,
           $6                       := DB6.DBD 304);
M001: NOP   0;
NETWORK
TITLE =
      A     M 0.0;
      =     L 0.0;
      BLD   103;
      A     M 0.1;
      JNB   M002;
      CALL  FC 105 (
           $1                       := P#P 260.0,
           $2                       := L#1101004800,
           $3                       := L#1082130432,
           $4                       := L 0.0,
           $5                       := DB6.DBW 298,
           $6                       := DB6.DBD 308);
M002: NOP   0;
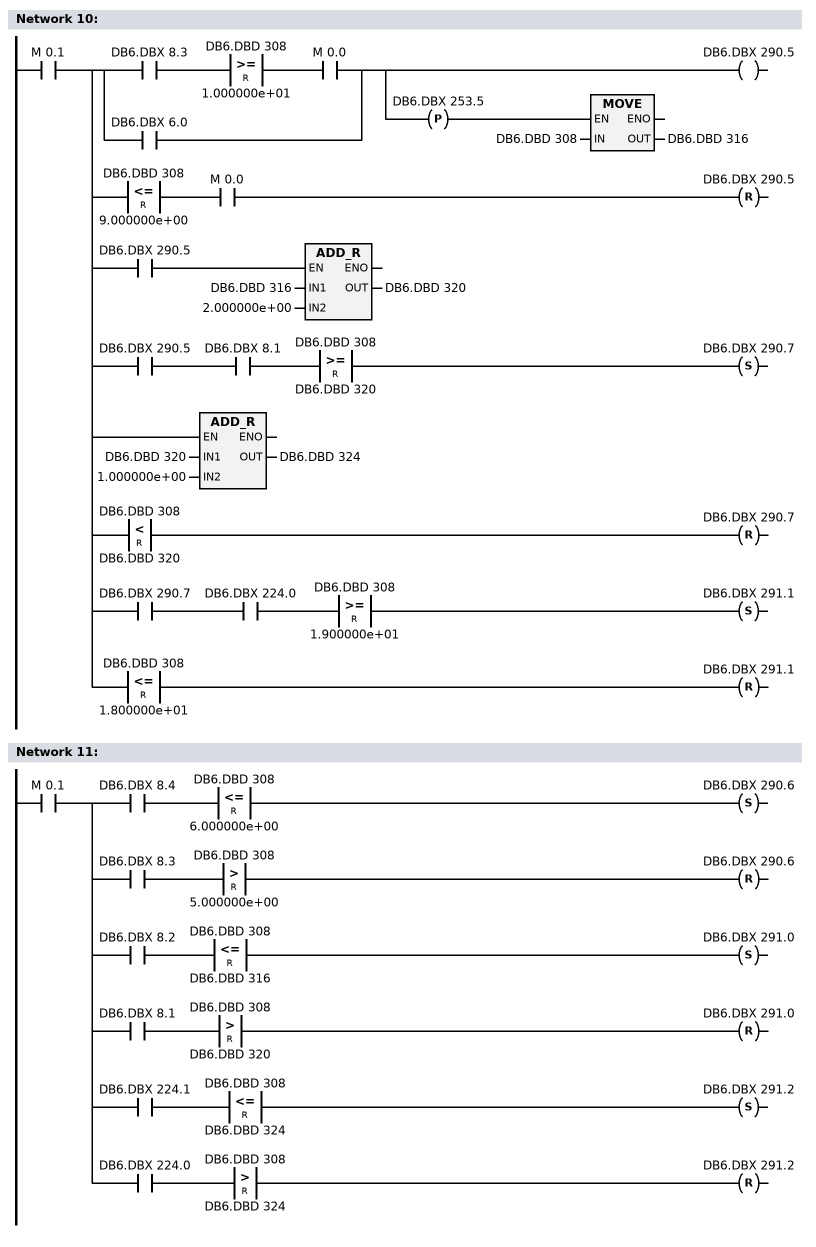
NETWORK
TITLE =
      A     M 0.1;
      =     L 0.0;
      A     L 0.0;
      A(;
      A     DB6.DBX 8.3;
      A(;
      L     DB6.DBD 308;
      L     1.000000e+01;
      >=R;
      );
      A     M 0.0;
      O     DB6.DBX 6.0;
      );
      =     L 0.1;
      A     L 0.1;
      BLD   102;
      =     DB6.DBX 290.5;
      A     L 0.1;
      FP    DB6.DBX 253.5;
      JNB   M003;
      L     DB6.DBD 308;
      T     DB6.DBD 316;
M003: NOP   0;
      A     L 0.0;
      A(;
      L     DB6.DBD 308;
      L     9.000000e+00;
      <=R;
      );
      A     M 0.0;
      R     DB6.DBX 290.5;
      A     L 0.0;
      A     DB6.DBX 290.5;
      JNB   M004;
      L     DB6.DBD 316;
      L     2.000000e+00;
      +R;
      T     DB6.DBD 320;
M004: NOP   0;
      A     L 0.0;
      A     DB6.DBX 290.5;
      A     DB6.DBX 8.1;
      A(;
      L     DB6.DBD 308;
      L     DB6.DBD 320;
      >=R;
      );
      S     DB6.DBX 290.7;
      A     L 0.0;
      JNB   M005;
      L     DB6.DBD 320;
      L     1.000000e+00;
      +R;
      T     DB6.DBD 324;
M005: NOP   0;
      A     L 0.0;
      A(;
      L     DB6.DBD 308;
      L     DB6.DBD 320;
      <R;
      );
      R     DB6.DBX 290.7;
      A     L 0.0;
      A     DB6.DBX 290.7;
      A     DB6.DBX 224.0;
      A(;
      L     DB6.DBD 308;
      L     1.900000e+01;
      >=R;
      );
      S     DB6.DBX 291.1;
      A     L 0.0;
      A(;
      L     DB6.DBD 308;
      L     1.800000e+01;
      <=R;
      );
      R     DB6.DBX 291.1;
NETWORK
TITLE =
      A     M 0.1;
      =     L 0.0;
      A     L 0.0;
      A     DB6.DBX 8.4;
      A(;
      L     DB6.DBD 308;
      L     6.000000e+00;
      <=R;
      );
      S     DB6.DBX 290.6;
      A     L 0.0;
      A     DB6.DBX 8.3;
      A(;
      L     DB6.DBD 308;
      L     5.000000e+00;
      >R;
      );
      R     DB6.DBX 290.6;
      A     L 0.0;
      A     DB6.DBX 8.2;
      A(;
      L     DB6.DBD 308;
      L     DB6.DBD 316;
      <=R;
      );
      S     DB6.DBX 291.0;
      A     L 0.0;
      A     DB6.DBX 8.1;
      A(;
      L     DB6.DBD 308;
      L     DB6.DBD 320;
      >R;
      );
      R     DB6.DBX 291.0;
      A     L 0.0;
      A     DB6.DBX 224.1;
      A(;
      L     DB6.DBD 308;
      L     DB6.DBD 324;
      <=R;
      );
      S     DB6.DBX 291.2;
      A     L 0.0;
      A     DB6.DBX 224.0;
      A(;
      L     DB6.DBD 308;
      L     DB6.DBD 324;
      >R;
      );
      R     DB6.DBX 291.2;
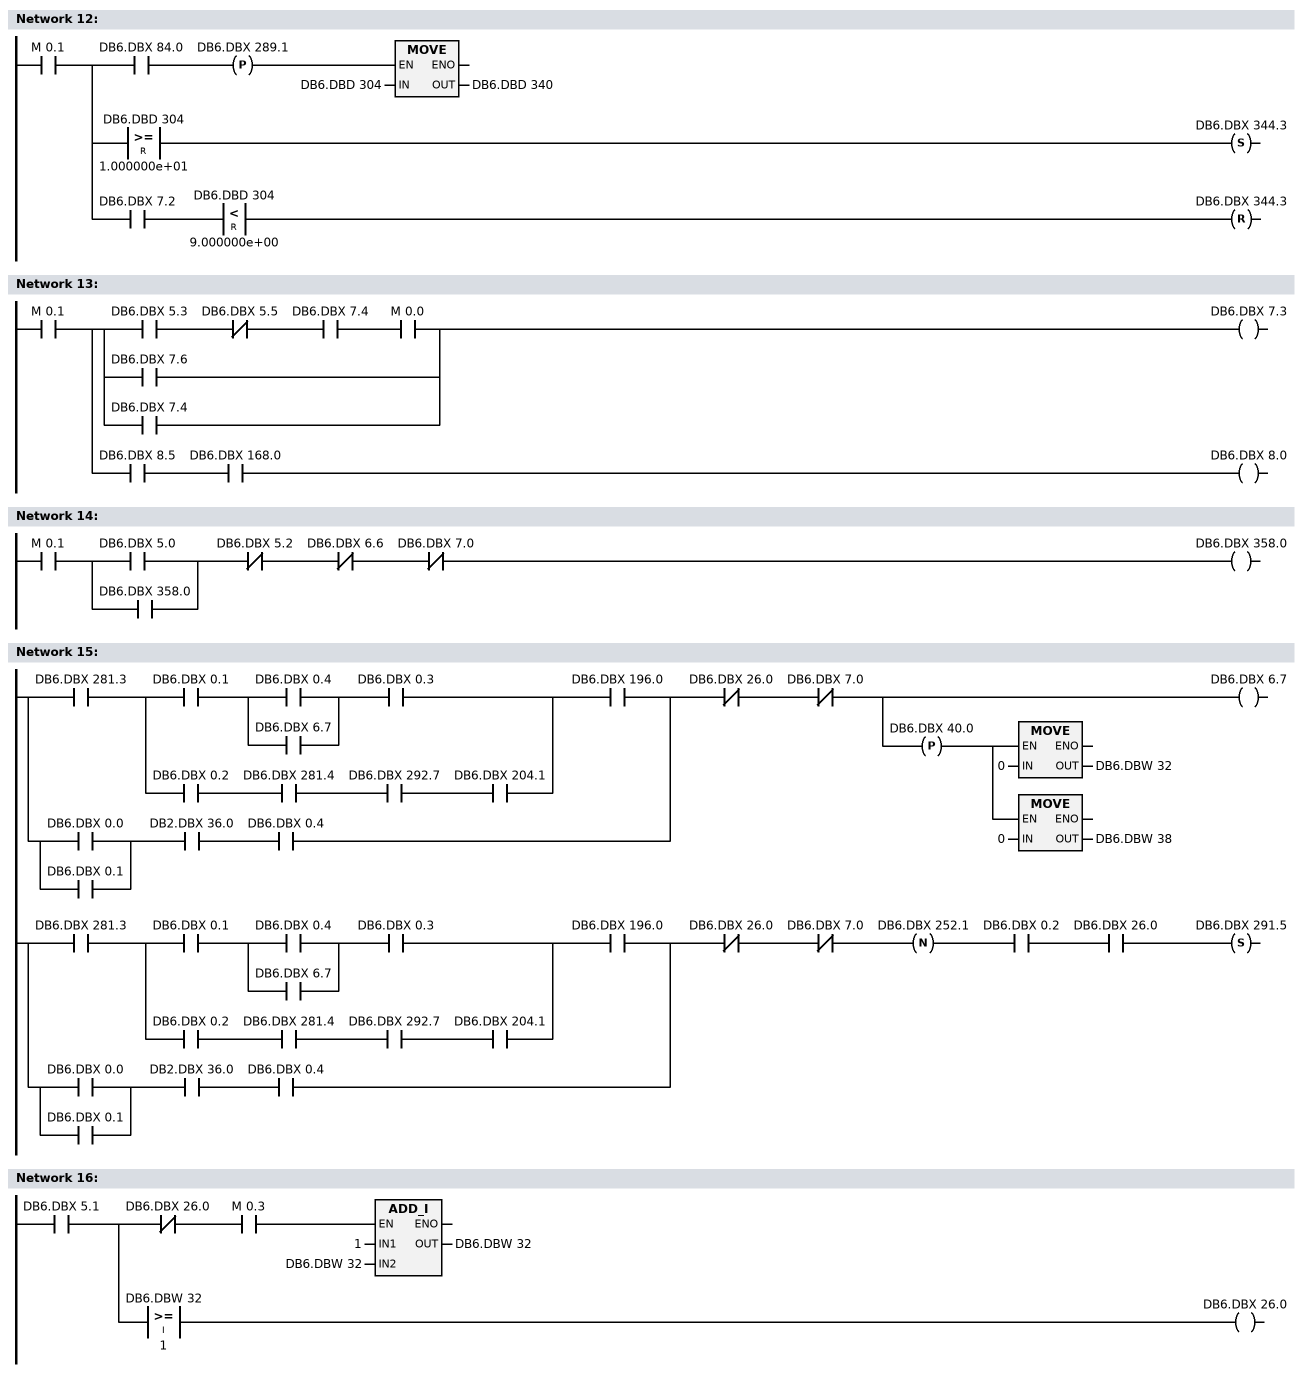
NETWORK
TITLE =
      A     M 0.1;
      =     L 0.0;
      A     L 0.0;
      A     DB6.DBX 84.0;
      FP    DB6.DBX 289.1;
      JNB   M006;
      L     DB6.DBD 304;
      T     DB6.DBD 340;
M006: NOP   0;
      A     L 0.0;
      A(;
      L     DB6.DBD 304;
      L     1.000000e+01;
      >=R;
      );
      S     DB6.DBX 344.3;
      A     L 0.0;
      A     DB6.DBX 7.2;
      A(;
      L     DB6.DBD 304;
      L     9.000000e+00;
      <R;
      );
      R     DB6.DBX 344.3;
NETWORK
TITLE =
      A     M 0.1;
      =     L 0.0;
      A     L 0.0;
      A(;
      A     DB6.DBX 5.3;
      AN    DB6.DBX 5.5;
      A     DB6.DBX 7.4;
      A     M 0.0;
      O     DB6.DBX 7.6;
      O     DB6.DBX 7.4;
      );
      =     DB6.DBX 7.3;
      A     L 0.0;
      A     DB6.DBX 8.5;
      A     DB6.DBX 168.0;
      =     DB6.DBX 8.0;
NETWORK
TITLE =
      A     M 0.1;
      A(;
      O     DB6.DBX 5.0;
      O     DB6.DBX 358.0;
      );
      AN    DB6.DBX 5.2;
      AN    DB6.DBX 6.6;
      AN    DB6.DBX 7.0;
      =     DB6.DBX 358.0;
NETWORK
TITLE =
      A(;
      A     DB6.DBX 281.3;
      A(;
      A     DB6.DBX 0.1;
      A(;
      O     DB6.DBX 0.4;
      O     DB6.DBX 6.7;
      );
      A     DB6.DBX 0.3;
      O;
      A     DB6.DBX 0.2;
      A     DB6.DBX 281.4;
      A     DB6.DBX 292.7;
      A     DB6.DBX 204.1;
      );
      A     DB6.DBX 196.0;
      O;
      A(;
      O     DB6.DBX 0.0;
      O     DB6.DBX 0.1;
      );
      A     DB2.DBX 36.0;
      A     DB6.DBX 0.4;
      );
      AN    DB6.DBX 26.0;
      AN    DB6.DBX 7.0;
      =     L 0.0;
      A     L 0.0;
      BLD   102;
      =     DB6.DBX 6.7;
      A(;
      A     L 0.0;
      FN    DB6.DBX 252.1;
      );
      A     DB6.DBX 0.2;
      A     DB6.DBX 26.0;
      S     DB6.DBX 291.5;
      A     L 0.0;
      FP    DB6.DBX 40.0;
      =     L 0.1;
      A     L 0.1;
      JNB   M007;
      L     0;
      T     DB6.DBW 32;
M007: NOP   0;
      A     L 0.1;
      JNB   M008;
      L     0;
      T     DB6.DBW 38;
M008: NOP   0;
NETWORK
TITLE =
      A     DB6.DBX 5.1;
      =     L 0.0;
      A     L 0.0;
      AN    DB6.DBX 26.0;
      A     M 0.3;
      JNB   M009;
      L     1;
      L     DB6.DBW 32;
      +I;
      T     DB6.DBW 32;
M009: NOP   0;
      A     L 0.0;
      A(;
      L     DB6.DBW 32;
      L     1;
      >=I;
      );
      =     DB6.DBX 26.0;
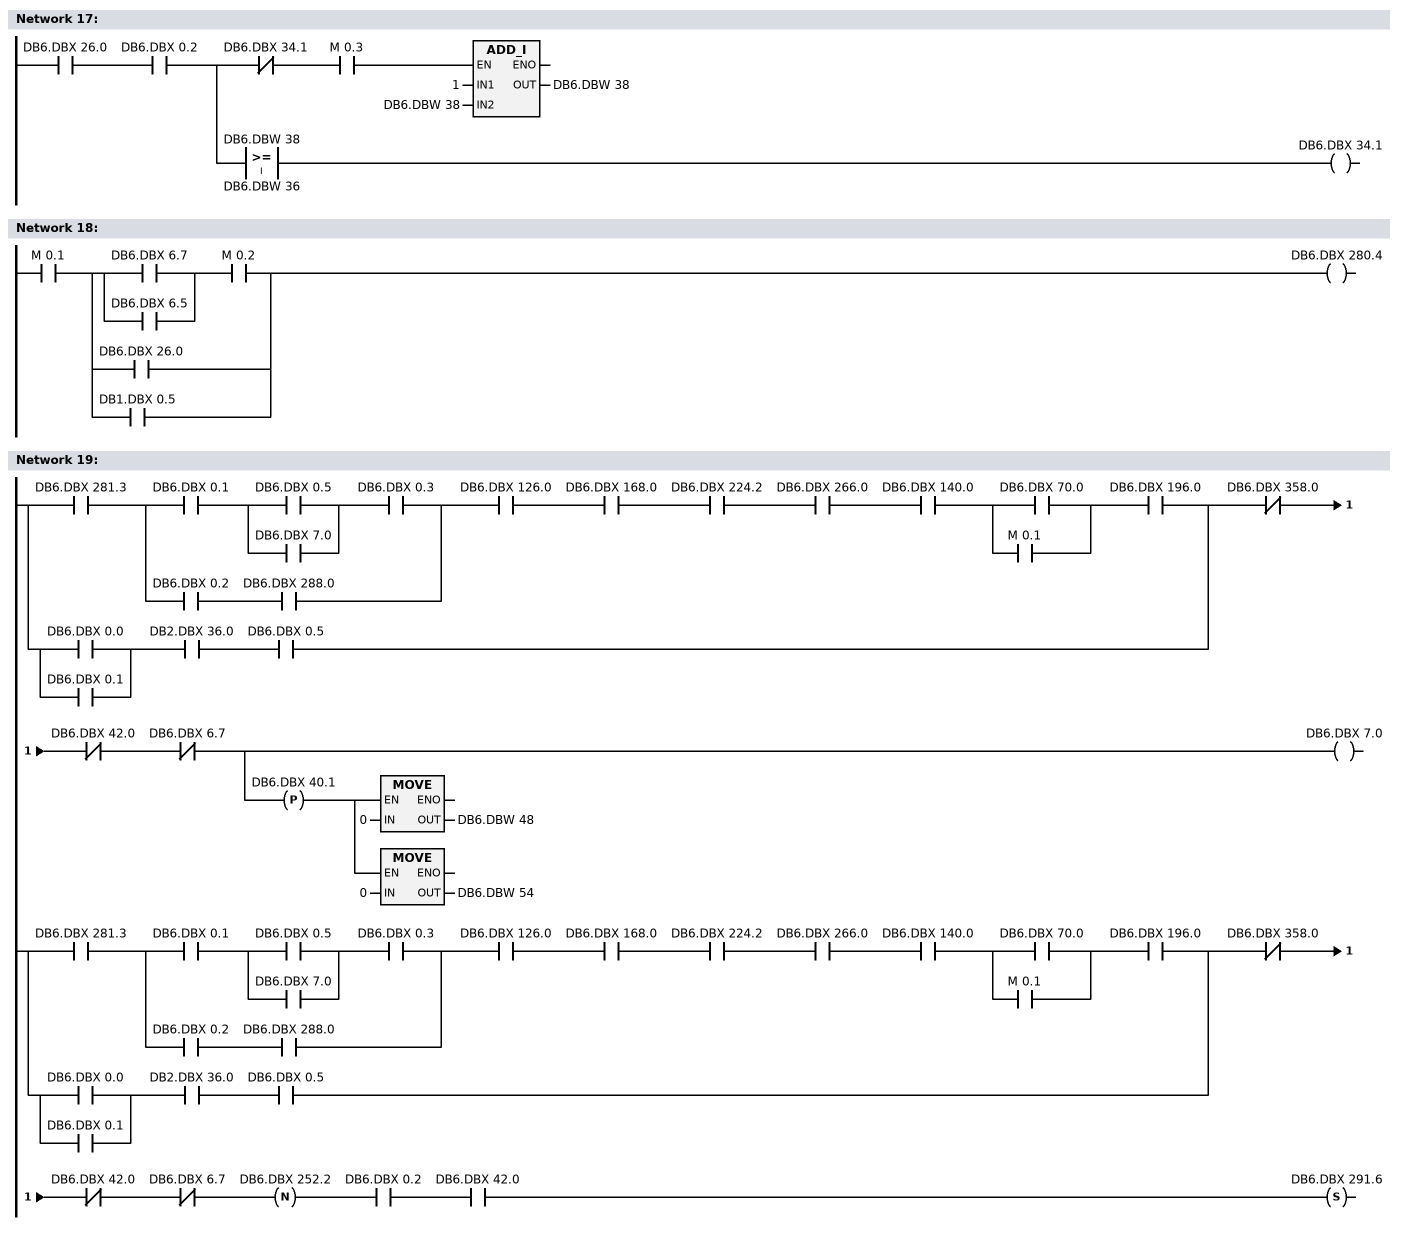
NETWORK
TITLE =
      A     DB6.DBX 26.0;
      A     DB6.DBX 0.2;
      =     L 0.0;
      A     L 0.0;
      AN    DB6.DBX 34.1;
      A     M 0.3;
      JNB   M010;
      L     1;
      L     DB6.DBW 38;
      +I;
      T     DB6.DBW 38;
M010: NOP   0;
      A     L 0.0;
      A(;
      L     DB6.DBW 38;
      L     DB6.DBW 36;
      >=I;
      );
      =     DB6.DBX 34.1;
NETWORK
TITLE =
      A     M 0.1;
      A(;
      A(;
      O     DB6.DBX 6.7;
      O     DB6.DBX 6.5;
      );
      A     M 0.2;
      O     DB6.DBX 26.0;
      O     DB1.DBX 0.5;
      );
      =     DB6.DBX 280.4;
NETWORK
TITLE =
      A(;
      A     DB6.DBX 281.3;
      A(;
      A     DB6.DBX 0.1;
      A(;
      O     DB6.DBX 0.5;
      O     DB6.DBX 7.0;
      );
      A     DB6.DBX 0.3;
      O;
      A     DB6.DBX 0.2;
      A     DB6.DBX 288.0;
      );
      A     DB6.DBX 126.0;
      A     DB6.DBX 168.0;
      A     DB6.DBX 224.2;
      A     DB6.DBX 266.0;
      A     DB6.DBX 140.0;
      A(;
      O     DB6.DBX 70.0;
      O     M 0.1;
      );
      A     DB6.DBX 196.0;
      O;
      A(;
      O     DB6.DBX 0.0;
      O     DB6.DBX 0.1;
      );
      A     DB2.DBX 36.0;
      A     DB6.DBX 0.5;
      );
      AN    DB6.DBX 358.0;
      AN    DB6.DBX 42.0;
      AN    DB6.DBX 6.7;
      =     L 0.0;
      A     L 0.0;
      BLD   102;
      =     DB6.DBX 7.0;
      A(;
      A     L 0.0;
      FN    DB6.DBX 252.2;
      );
      A     DB6.DBX 0.2;
      A     DB6.DBX 42.0;
      S     DB6.DBX 291.6;
      A     L 0.0;
      FP    DB6.DBX 40.1;
      =     L 0.1;
      A     L 0.1;
      JNB   M011;
      L     0;
      T     DB6.DBW 48;
M011: NOP   0;
      A     L 0.1;
      JNB   M012;
      L     0;
      T     DB6.DBW 54;
M012: NOP   0;
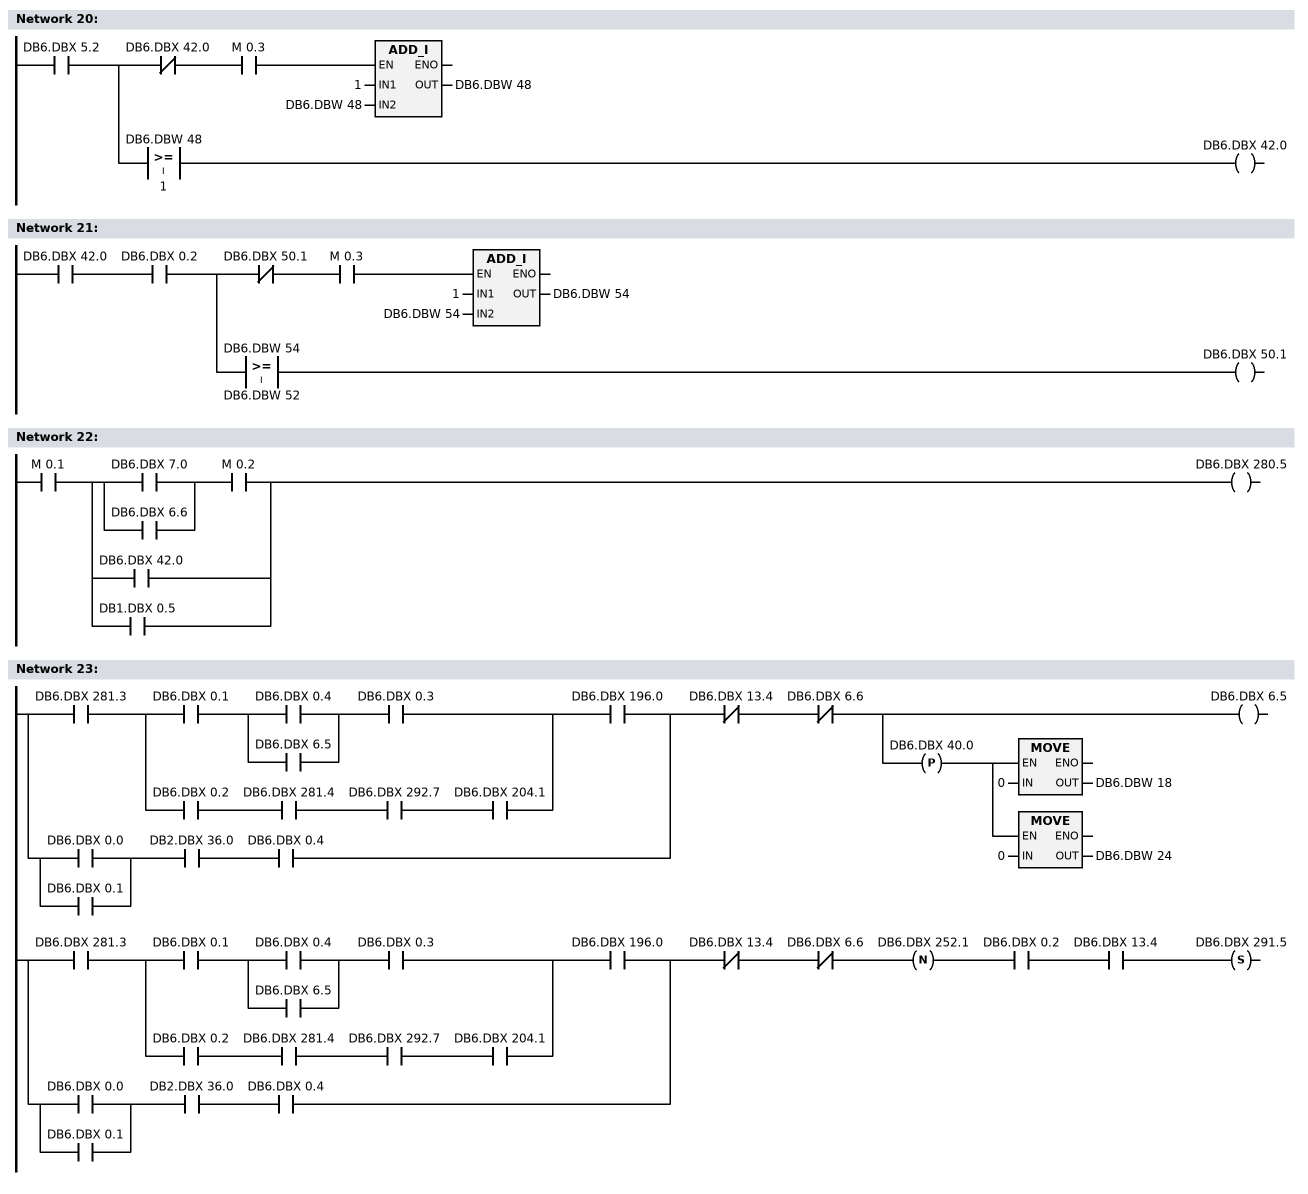
NETWORK
TITLE =
      A     DB6.DBX 5.2;
      =     L 0.0;
      A     L 0.0;
      AN    DB6.DBX 42.0;
      A     M 0.3;
      JNB   M013;
      L     1;
      L     DB6.DBW 48;
      +I;
      T     DB6.DBW 48;
M013: NOP   0;
      A     L 0.0;
      A(;
      L     DB6.DBW 48;
      L     1;
      >=I;
      );
      =     DB6.DBX 42.0;
NETWORK
TITLE =
      A     DB6.DBX 42.0;
      A     DB6.DBX 0.2;
      =     L 0.0;
      A     L 0.0;
      AN    DB6.DBX 50.1;
      A     M 0.3;
      JNB   M014;
      L     1;
      L     DB6.DBW 54;
      +I;
      T     DB6.DBW 54;
M014: NOP   0;
      A     L 0.0;
      A(;
      L     DB6.DBW 54;
      L     DB6.DBW 52;
      >=I;
      );
      =     DB6.DBX 50.1;
NETWORK
TITLE =
      A     M 0.1;
      A(;
      A(;
      O     DB6.DBX 7.0;
      O     DB6.DBX 6.6;
      );
      A     M 0.2;
      O     DB6.DBX 42.0;
      O     DB1.DBX 0.5;
      );
      =     DB6.DBX 280.5;
NETWORK
TITLE =
      A(;
      A     DB6.DBX 281.3;
      A(;
      A     DB6.DBX 0.1;
      A(;
      O     DB6.DBX 0.4;
      O     DB6.DBX 6.5;
      );
      A     DB6.DBX 0.3;
      O;
      A     DB6.DBX 0.2;
      A     DB6.DBX 281.4;
      A     DB6.DBX 292.7;
      A     DB6.DBX 204.1;
      );
      A     DB6.DBX 196.0;
      O;
      A(;
      O     DB6.DBX 0.0;
      O     DB6.DBX 0.1;
      );
      A     DB2.DBX 36.0;
      A     DB6.DBX 0.4;
      );
      AN    DB6.DBX 13.4;
      AN    DB6.DBX 6.6;
      =     L 0.0;
      A     L 0.0;
      BLD   102;
      =     DB6.DBX 6.5;
      A(;
      A     L 0.0;
      FN    DB6.DBX 252.1;
      );
      A     DB6.DBX 0.2;
      A     DB6.DBX 13.4;
      S     DB6.DBX 291.5;
      A     L 0.0;
      FP    DB6.DBX 40.0;
      =     L 0.1;
      A     L 0.1;
      JNB   M015;
      L     0;
      T     DB6.DBW 18;
M015: NOP   0;
      A     L 0.1;
      JNB   M016;
      L     0;
      T     DB6.DBW 24;
M016: NOP   0;
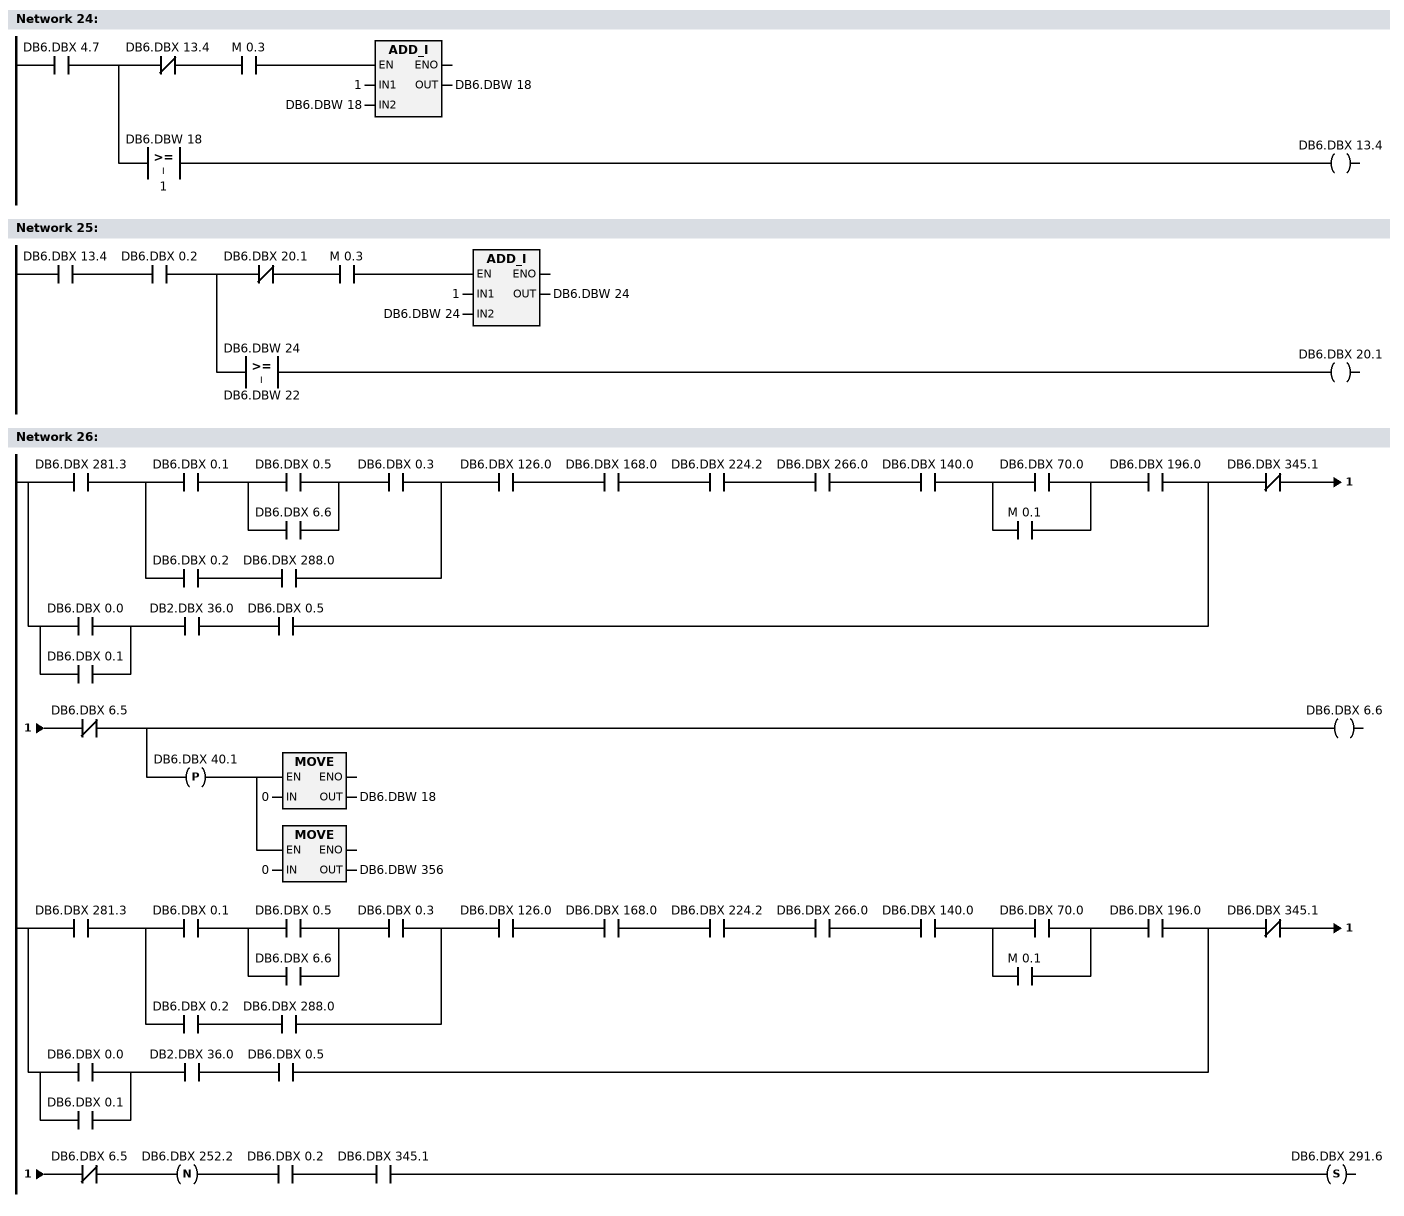
NETWORK
TITLE =
      A     DB6.DBX 4.7;
      =     L 0.0;
      A     L 0.0;
      AN    DB6.DBX 13.4;
      A     M 0.3;
      JNB   M017;
      L     1;
      L     DB6.DBW 18;
      +I;
      T     DB6.DBW 18;
M017: NOP   0;
      A     L 0.0;
      A(;
      L     DB6.DBW 18;
      L     1;
      >=I;
      );
      =     DB6.DBX 13.4;
NETWORK
TITLE =
      A     DB6.DBX 13.4;
      A     DB6.DBX 0.2;
      =     L 0.0;
      A     L 0.0;
      AN    DB6.DBX 20.1;
      A     M 0.3;
      JNB   M018;
      L     1;
      L     DB6.DBW 24;
      +I;
      T     DB6.DBW 24;
M018: NOP   0;
      A     L 0.0;
      A(;
      L     DB6.DBW 24;
      L     DB6.DBW 22;
      >=I;
      );
      =     DB6.DBX 20.1;
NETWORK
TITLE =
      A(;
      A     DB6.DBX 281.3;
      A(;
      A     DB6.DBX 0.1;
      A(;
      O     DB6.DBX 0.5;
      O     DB6.DBX 6.6;
      );
      A     DB6.DBX 0.3;
      O;
      A     DB6.DBX 0.2;
      A     DB6.DBX 288.0;
      );
      A     DB6.DBX 126.0;
      A     DB6.DBX 168.0;
      A     DB6.DBX 224.2;
      A     DB6.DBX 266.0;
      A     DB6.DBX 140.0;
      A(;
      O     DB6.DBX 70.0;
      O     M 0.1;
      );
      A     DB6.DBX 196.0;
      O;
      A(;
      O     DB6.DBX 0.0;
      O     DB6.DBX 0.1;
      );
      A     DB2.DBX 36.0;
      A     DB6.DBX 0.5;
      );
      AN    DB6.DBX 345.1;
      AN    DB6.DBX 6.5;
      =     L 0.0;
      A     L 0.0;
      BLD   102;
      =     DB6.DBX 6.6;
      A(;
      A     L 0.0;
      FN    DB6.DBX 252.2;
      );
      A     DB6.DBX 0.2;
      A     DB6.DBX 345.1;
      S     DB6.DBX 291.6;
      A     L 0.0;
      FP    DB6.DBX 40.1;
      =     L 0.1;
      A     L 0.1;
      JNB   M019;
      L     0;
      T     DB6.DBW 18;
M019: NOP   0;
      A     L 0.1;
      JNB   M020;
      L     0;
      T     DB6.DBW 356;
M020: NOP   0;
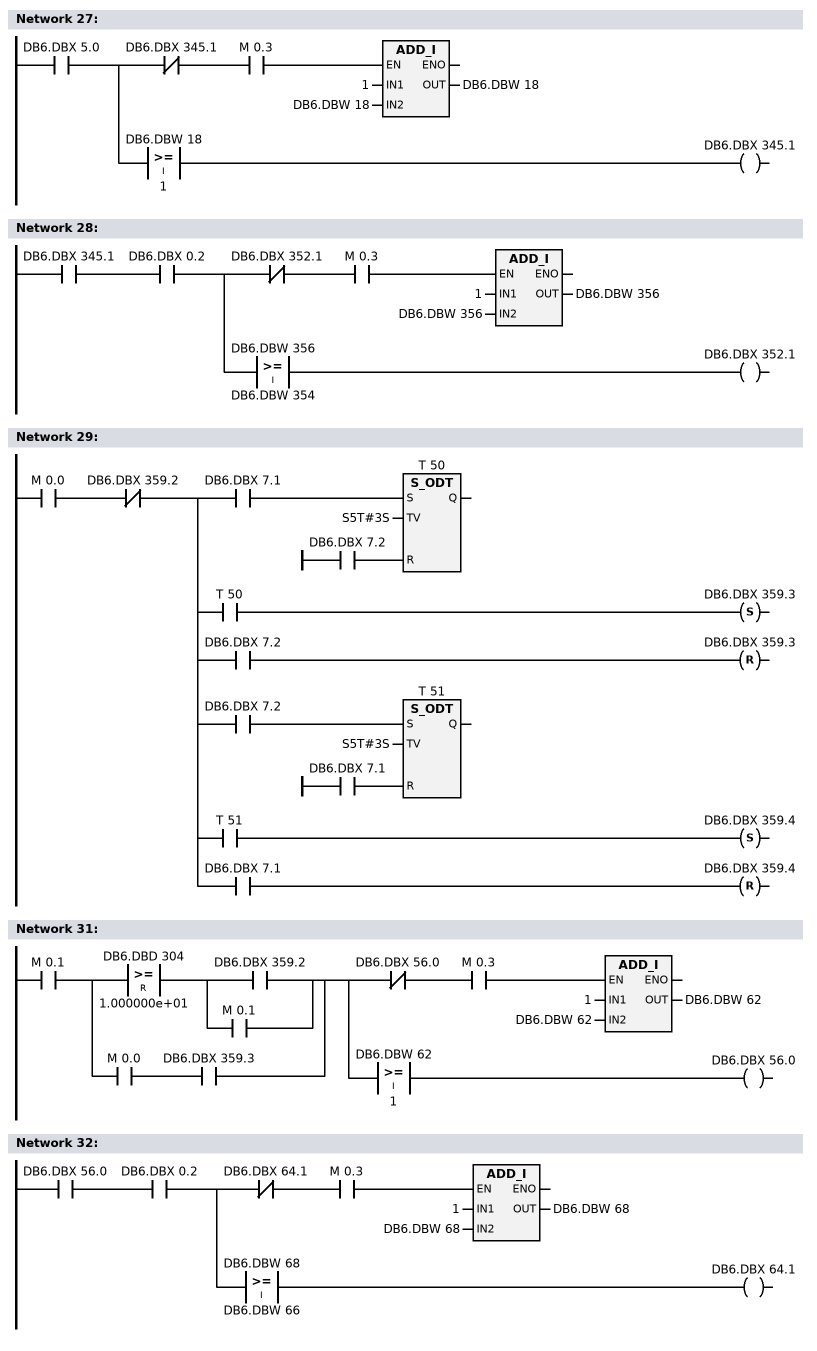
NETWORK
TITLE =
      A     DB6.DBX 5.0;
      =     L 0.0;
      A     L 0.0;
      AN    DB6.DBX 345.1;
      A     M 0.3;
      JNB   M021;
      L     1;
      L     DB6.DBW 18;
      +I;
      T     DB6.DBW 18;
M021: NOP   0;
      A     L 0.0;
      A(;
      L     DB6.DBW 18;
      L     1;
      >=I;
      );
      =     DB6.DBX 345.1;
NETWORK
TITLE =
      A     DB6.DBX 345.1;
      A     DB6.DBX 0.2;
      =     L 0.0;
      A     L 0.0;
      AN    DB6.DBX 352.1;
      A     M 0.3;
      JNB   M022;
      L     1;
      L     DB6.DBW 356;
      +I;
      T     DB6.DBW 356;
M022: NOP   0;
      A     L 0.0;
      A(;
      L     DB6.DBW 356;
      L     DB6.DBW 354;
      >=I;
      );
      =     DB6.DBX 352.1;
NETWORK
TITLE =
      A     M 0.0;
      AN    DB6.DBX 359.2;
      =     L 0.0;
      A     L 0.0;
      A     DB6.DBX 7.1;
      L     S5T#3S;
      SD    T 50;
      A     DB6.DBX 7.2;
      R     T 50;
      NOP   0;
      NOP   0;
      NOP   0;
      A     L 0.0;
      A     T 50;
      S     DB6.DBX 359.3;
      A     L 0.0;
      A     DB6.DBX 7.2;
      R     DB6.DBX 359.3;
      A     L 0.0;
      A     DB6.DBX 7.2;
      L     S5T#3S;
      SD    T 51;
      A     DB6.DBX 7.1;
      R     T 51;
      NOP   0;
      NOP   0;
      NOP   0;
      A     L 0.0;
      A     T 51;
      S     DB6.DBX 359.4;
      A     L 0.0;
      A     DB6.DBX 7.1;
      R     DB6.DBX 359.4;
NETWORK
TITLE =
      A(;
      A     DB6.DBX 281.3;
      A(;
      A     DB6.DBX 0.1;
      A(;
      O     DB6.DBX 0.6;
      O     DB6.DBX 7.1;
      );
      A     DB6.DBX 0.3;
      O;
      A     DB6.DBX 0.2;
      A(;
      A     DB6.DBX 281.4;
      A(;
      ON    DB6.DBX 291.7;
      O     M 0.1;
      );
      O;
      A     DB6.DBX 288.0;
      A     DB6.DBX 293.0;
      A(;
      ON    DB6.DBX 291.7;
      O     M 0.1;
      );
      );
      );
      A(;
      A     DB6.DBX 42.0;
      A     DB6.DBX 182.0;
      A     DB6.DBX 154.0;
      A     DB6.DBX 253.6;
      A     DB6.DBX 238.0;
      O;
      A     DB6.DBX 42.0;
      A     DB6.DBX 126.0;
      A     DB6.DBX 168.0;
      A     DB6.DBX 224.2;
      A     DB6.DBX 266.0;
      A     DB6.DBX 140.0;
      A     DB6.DBX 210.0;
      );
      O;
      A(;
      O     DB6.DBX 0.0;
      O     DB6.DBX 0.1;
      );
      A     DB2.DBX 36.0;
      A     DB6.DBX 0.6;
      );
      AN    DB6.DBX 56.0;
      AN    DB6.DBX 7.2;
      =     L 0.0;
      A     L 0.0;
      AN    DB6.DBX 0.2;
      =     L 0.1;
      A     L 0.1;
      BLD   102;
      =     DB6.DBX 7.1;
      A(;
      A     L 0.1;
      FN    DB6.DBX 252.3;
      );
      A     DB6.DBX 56.0;
      A     DB6.DBX 0.2;
      S     DB6.DBX 291.7;
      A     L 0.0;
      FP    DB6.DBX 40.2;
      =     L 0.1;
      A     L 0.1;
      A     DB6.DBX 0.2;
      S     DB6.DBX 291.7;
      A     L 0.1;
      JNB   M023;
      L     0;
      T     DB6.DBW 62;
M023: NOP   0;
      A     L 0.1;
      JNB   M024;
      L     0;
      T     DB6.DBW 68;
M024: NOP   0;
NETWORK
TITLE =
      A     M 0.1;
      A(;
      A(;
      L     DB6.DBD 304;
      L     1.000000e+01;
      >=R;
      );
      A(;
      O     DB6.DBX 359.2;
      O     M 0.1;
      );
      O;
      A     M 0.0;
      A     DB6.DBX 359.3;
      );
      =     L 0.0;
      A     L 0.0;
      AN    DB6.DBX 56.0;
      A     M 0.3;
      JNB   M025;
      L     1;
      L     DB6.DBW 62;
      +I;
      T     DB6.DBW 62;
M025: NOP   0;
      A     L 0.0;
      A(;
      L     DB6.DBW 62;
      L     1;
      >=I;
      );
      =     DB6.DBX 56.0;
NETWORK
TITLE =
      A     DB6.DBX 56.0;
      A     DB6.DBX 0.2;
      =     L 0.0;
      A     L 0.0;
      AN    DB6.DBX 64.1;
      A     M 0.3;
      JNB   M026;
      L     1;
      L     DB6.DBW 68;
      +I;
      T     DB6.DBW 68;
M026: NOP   0;
      A     L 0.0;
      A(;
      L     DB6.DBW 68;
      L     DB6.DBW 66;
      >=I;
      );
      =     DB6.DBX 64.1;
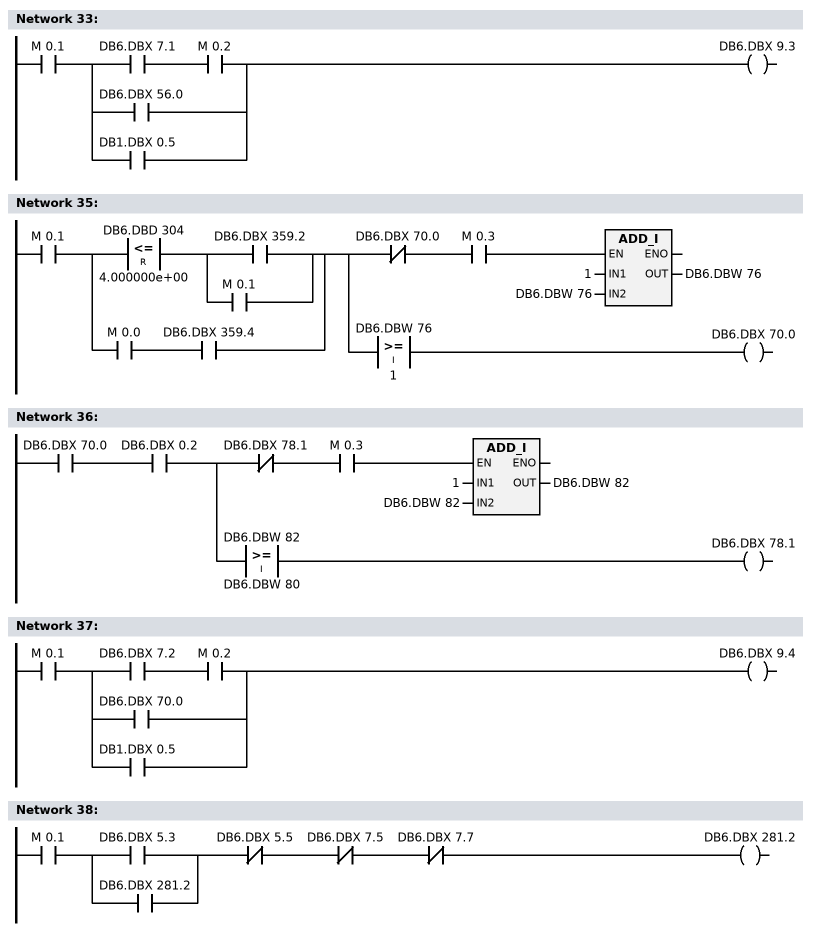
NETWORK
TITLE =
      A     M 0.1;
      A(;
      A     DB6.DBX 7.1;
      A     M 0.2;
      O     DB6.DBX 56.0;
      O     DB1.DBX 0.5;
      );
      =     DB6.DBX 9.3;
NETWORK
TITLE =
      A(;
      A     DB6.DBX 281.3;
      A(;
      A     DB6.DBX 0.1;
      A(;
      O     DB6.DBX 0.7;
      O     DB6.DBX 7.2;
      );
      A     DB6.DBX 0.3;
      O;
      A     DB6.DBX 0.2;
      A(;
      A     DB6.DBX 281.4;
      A     DB6.DBX 292.2;
      A     DB6.DBX 134.1;
      O;
      A     DB6.DBX 288.0;
      A     DB6.DBX 292.2;
      A     DB6.DBX 134.1;
      );
      );
      A(;
      A     DB6.DBX 42.0;
      A     DB6.DBX 126.0;
      A     DB6.DBX 168.0;
      A     DB6.DBX 224.2;
      A     DB6.DBX 266.0;
      A     DB6.DBX 140.0;
      O;
      A     DB6.DBX 42.0;
      A     DB6.DBX 126.0;
      A     DB6.DBX 182.0;
      A     DB6.DBX 238.0;
      A     DB6.DBX 253.6;
      A     DB6.DBX 154.0;
      A     DB6.DBX 210.0;
      );
      O;
      A(;
      O     DB6.DBX 0.0;
      O     DB6.DBX 0.1;
      );
      A     DB2.DBX 36.0;
      A     DB6.DBX 0.7;
      );
      AN    DB6.DBX 70.0;
      AN    DB6.DBX 7.1;
      =     L 0.0;
      A     L 0.0;
      AN    DB6.DBX 0.2;
      =     L 0.1;
      A     L 0.1;
      BLD   102;
      =     DB6.DBX 7.2;
      A(;
      A     L 0.1;
      FN    DB6.DBX 252.4;
      );
      A     DB6.DBX 0.2;
      A     DB6.DBX 70.0;
      S     DB6.DBX 292.0;
      A     L 0.0;
      FP    DB6.DBX 40.3;
      =     L 0.1;
      A     L 0.1;
      A     DB6.DBX 0.2;
      S     DB6.DBX 292.0;
      A     L 0.1;
      JNB   M027;
      L     0;
      T     DB6.DBW 76;
M027: NOP   0;
      A     L 0.1;
      JNB   M028;
      L     0;
      T     DB6.DBW 82;
M028: NOP   0;
NETWORK
TITLE =
      A     M 0.1;
      A(;
      A(;
      L     DB6.DBD 304;
      L     4.000000e+00;
      <=R;
      );
      A(;
      O     DB6.DBX 359.2;
      O     M 0.1;
      );
      O;
      A     M 0.0;
      A     DB6.DBX 359.4;
      );
      =     L 0.0;
      A     L 0.0;
      AN    DB6.DBX 70.0;
      A     M 0.3;
      JNB   M029;
      L     1;
      L     DB6.DBW 76;
      +I;
      T     DB6.DBW 76;
M029: NOP   0;
      A     L 0.0;
      A(;
      L     DB6.DBW 76;
      L     1;
      >=I;
      );
      =     DB6.DBX 70.0;
NETWORK
TITLE =
      A     DB6.DBX 70.0;
      A     DB6.DBX 0.2;
      =     L 0.0;
      A     L 0.0;
      AN    DB6.DBX 78.1;
      A     M 0.3;
      JNB   M030;
      L     1;
      L     DB6.DBW 82;
      +I;
      T     DB6.DBW 82;
M030: NOP   0;
      A     L 0.0;
      A(;
      L     DB6.DBW 82;
      L     DB6.DBW 80;
      >=I;
      );
      =     DB6.DBX 78.1;
NETWORK
TITLE =
      A     M 0.1;
      A(;
      A     DB6.DBX 7.2;
      A     M 0.2;
      O     DB6.DBX 70.0;
      O     DB1.DBX 0.5;
      );
      =     DB6.DBX 9.4;
NETWORK
TITLE =
      A     M 0.1;
      A(;
      O     DB6.DBX 5.3;
      O     DB6.DBX 281.2;
      );
      AN    DB6.DBX 5.5;
      AN    DB6.DBX 7.5;
      AN    DB6.DBX 7.7;
      =     DB6.DBX 281.2;
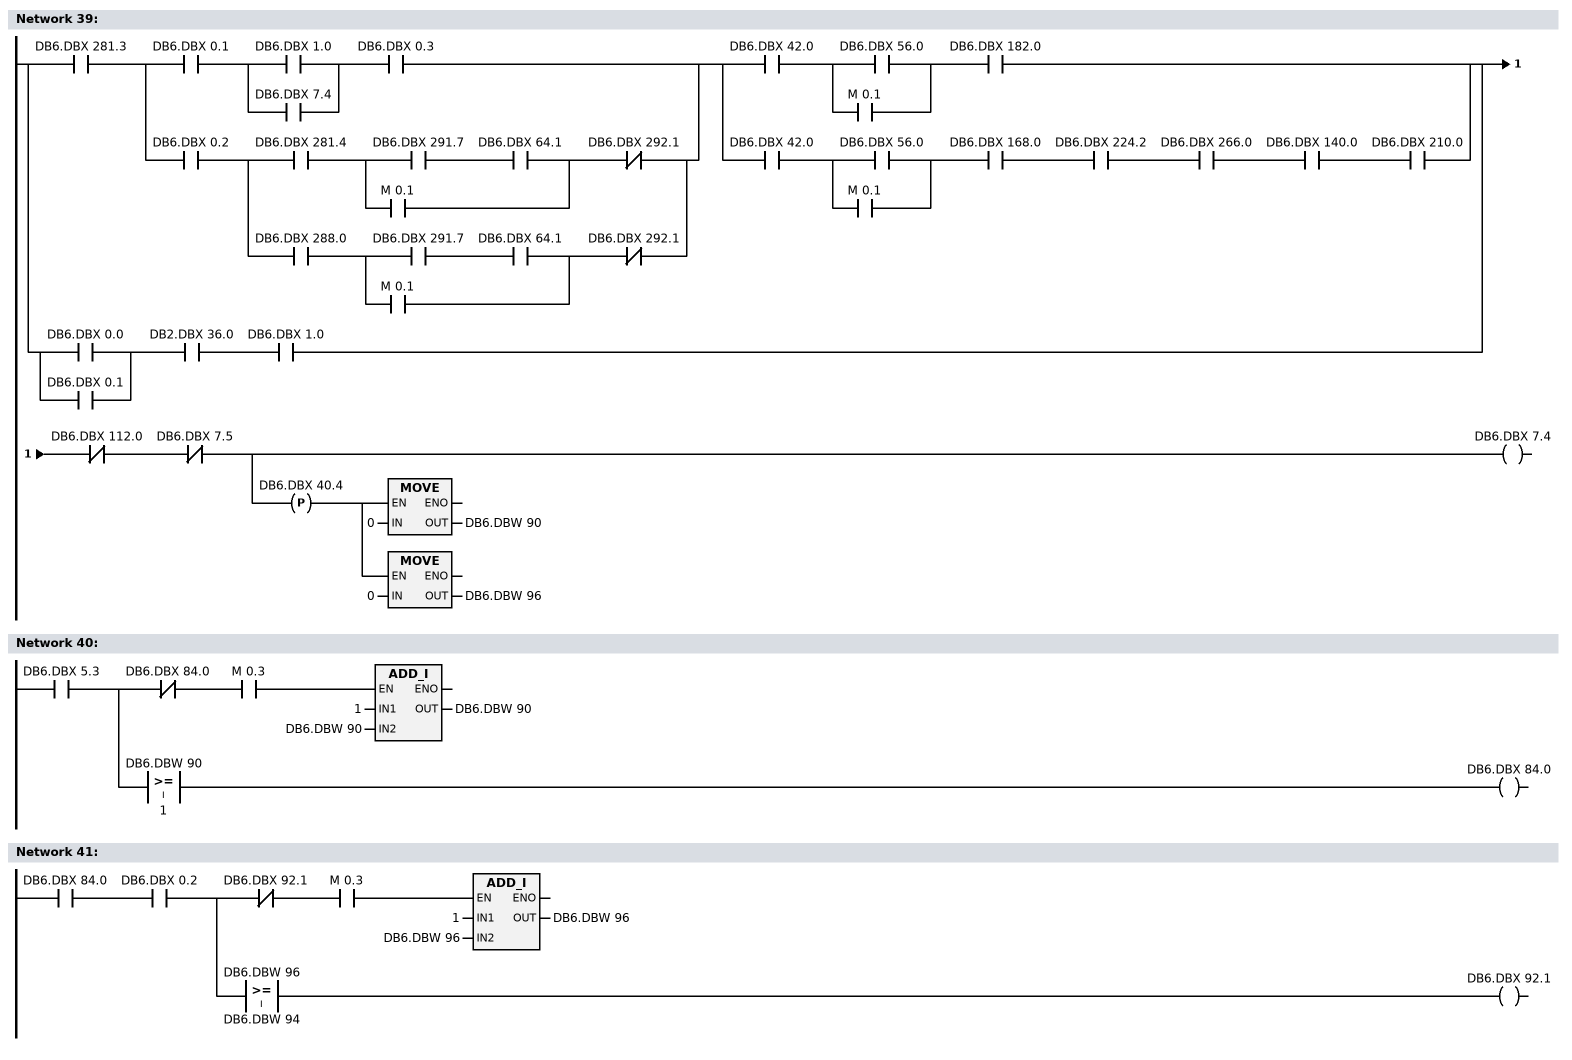
NETWORK
TITLE =
      A(;
      A     DB6.DBX 281.3;
      A(;
      A     DB6.DBX 0.1;
      A(;
      O     DB6.DBX 1.0;
      O     DB6.DBX 7.4;
      );
      A     DB6.DBX 0.3;
      O;
      A     DB6.DBX 0.2;
      A(;
      A     DB6.DBX 281.4;
      A(;
      A     DB6.DBX 291.7;
      A     DB6.DBX 64.1;
      O     M 0.1;
      );
      AN    DB6.DBX 292.1;
      O;
      A     DB6.DBX 288.0;
      A(;
      A     DB6.DBX 291.7;
      A     DB6.DBX 64.1;
      O     M 0.1;
      );
      AN    DB6.DBX 292.1;
      );
      );
      A(;
      A     DB6.DBX 42.0;
      A(;
      O     DB6.DBX 56.0;
      O     M 0.1;
      );
      A     DB6.DBX 182.0;
      O;
      A     DB6.DBX 42.0;
      A(;
      O     DB6.DBX 56.0;
      O     M 0.1;
      );
      A     DB6.DBX 168.0;
      A     DB6.DBX 224.2;
      A     DB6.DBX 266.0;
      A     DB6.DBX 140.0;
      A     DB6.DBX 210.0;
      );
      O;
      A(;
      O     DB6.DBX 0.0;
      O     DB6.DBX 0.1;
      );
      A     DB2.DBX 36.0;
      A     DB6.DBX 1.0;
      );
      AN    DB6.DBX 112.0;
      AN    DB6.DBX 7.5;
      =     L 0.0;
      A     L 0.0;
      BLD   102;
      =     DB6.DBX 7.4;
      A     L 0.0;
      FP    DB6.DBX 40.4;
      =     L 0.1;
      A     L 0.1;
      JNB   M031;
      L     0;
      T     DB6.DBW 90;
M031: NOP   0;
      A     L 0.1;
      JNB   M032;
      L     0;
      T     DB6.DBW 96;
M032: NOP   0;
NETWORK
TITLE =
      A     DB6.DBX 5.3;
      =     L 0.0;
      A     L 0.0;
      AN    DB6.DBX 84.0;
      A     M 0.3;
      JNB   M033;
      L     1;
      L     DB6.DBW 90;
      +I;
      T     DB6.DBW 90;
M033: NOP   0;
      A     L 0.0;
      A(;
      L     DB6.DBW 90;
      L     1;
      >=I;
      );
      =     DB6.DBX 84.0;
NETWORK
TITLE =
      A     DB6.DBX 84.0;
      A     DB6.DBX 0.2;
      =     L 0.0;
      A     L 0.0;
      AN    DB6.DBX 92.1;
      A     M 0.3;
      JNB   M034;
      L     1;
      L     DB6.DBW 96;
      +I;
      T     DB6.DBW 96;
M034: NOP   0;
      A     L 0.0;
      A(;
      L     DB6.DBW 96;
      L     DB6.DBW 94;
      >=I;
      );
      =     DB6.DBX 92.1;
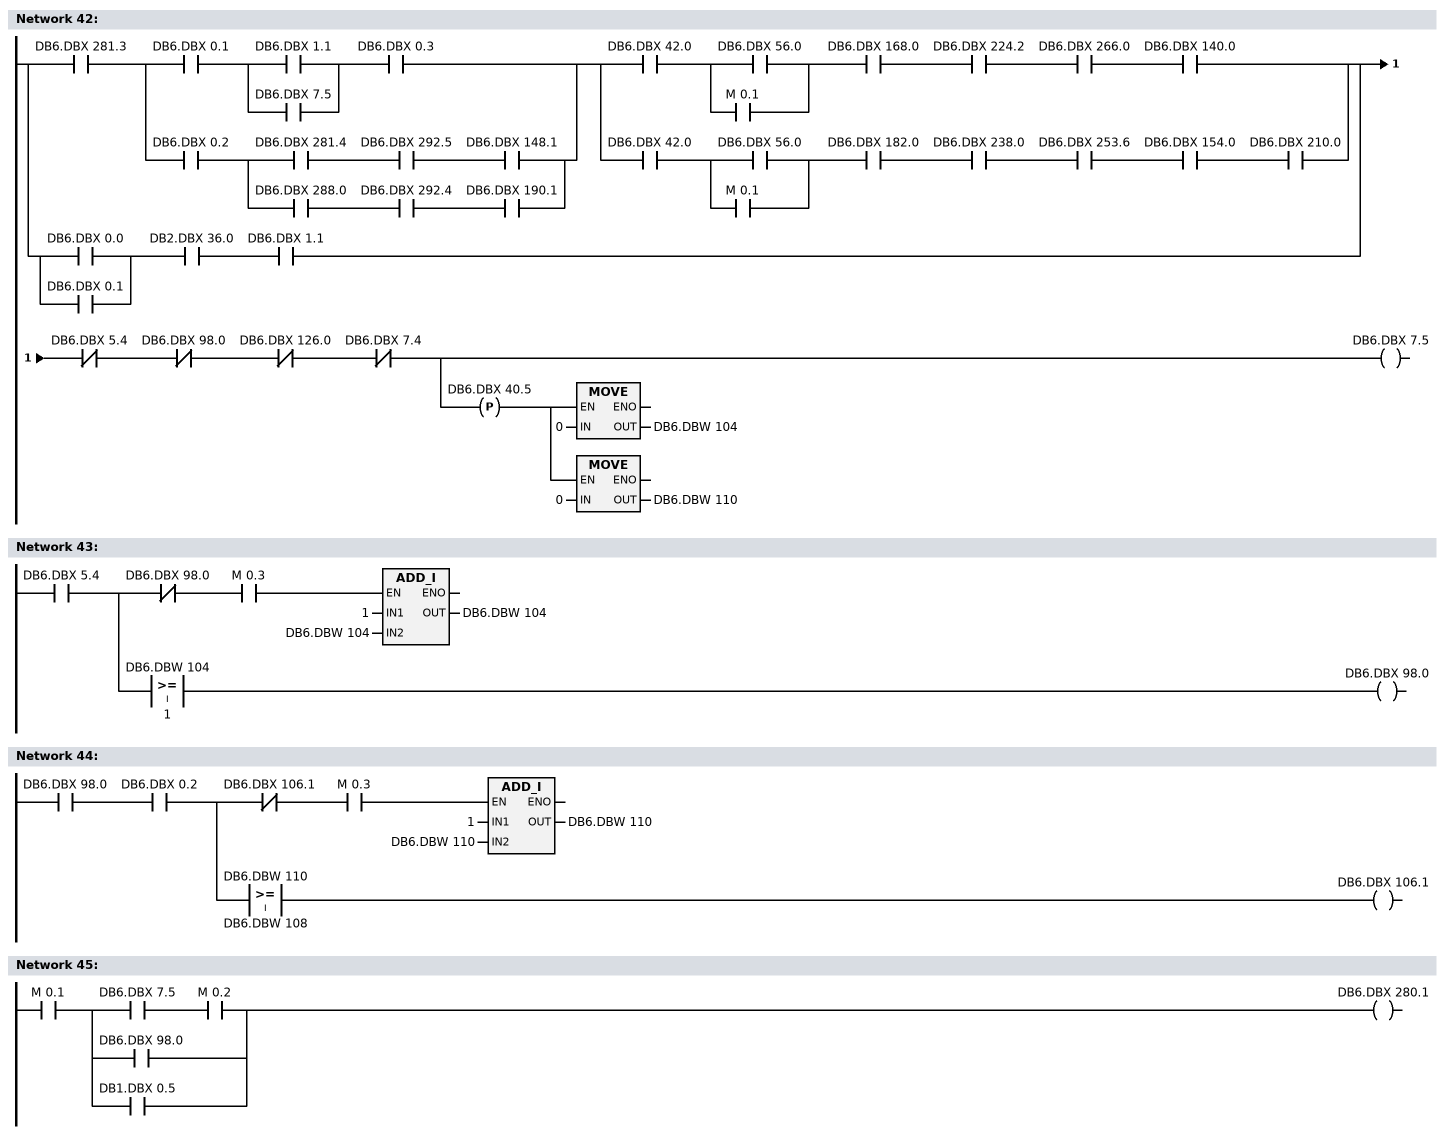
NETWORK
TITLE =
      A(;
      A     DB6.DBX 281.3;
      A(;
      A     DB6.DBX 0.1;
      A(;
      O     DB6.DBX 1.1;
      O     DB6.DBX 7.5;
      );
      A     DB6.DBX 0.3;
      O;
      A     DB6.DBX 0.2;
      A(;
      A     DB6.DBX 281.4;
      A     DB6.DBX 292.5;
      A     DB6.DBX 148.1;
      O;
      A     DB6.DBX 288.0;
      A     DB6.DBX 292.4;
      A     DB6.DBX 190.1;
      );
      );
      A(;
      A     DB6.DBX 42.0;
      A(;
      O     DB6.DBX 56.0;
      O     M 0.1;
      );
      A     DB6.DBX 168.0;
      A     DB6.DBX 224.2;
      A     DB6.DBX 266.0;
      A     DB6.DBX 140.0;
      O;
      A     DB6.DBX 42.0;
      A(;
      O     DB6.DBX 56.0;
      O     M 0.1;
      );
      A     DB6.DBX 182.0;
      A     DB6.DBX 238.0;
      A     DB6.DBX 253.6;
      A     DB6.DBX 154.0;
      A     DB6.DBX 210.0;
      );
      O;
      A(;
      O     DB6.DBX 0.0;
      O     DB6.DBX 0.1;
      );
      A     DB2.DBX 36.0;
      A     DB6.DBX 1.1;
      );
      AN    DB6.DBX 5.4;
      AN    DB6.DBX 98.0;
      AN    DB6.DBX 126.0;
      AN    DB6.DBX 7.4;
      =     L 0.0;
      A     L 0.0;
      BLD   102;
      =     DB6.DBX 7.5;
      A     L 0.0;
      FP    DB6.DBX 40.5;
      =     L 0.1;
      A     L 0.1;
      JNB   M035;
      L     0;
      T     DB6.DBW 104;
M035: NOP   0;
      A     L 0.1;
      JNB   M036;
      L     0;
      T     DB6.DBW 110;
M036: NOP   0;
NETWORK
TITLE =
      A     DB6.DBX 5.4;
      =     L 0.0;
      A     L 0.0;
      AN    DB6.DBX 98.0;
      A     M 0.3;
      JNB   M037;
      L     1;
      L     DB6.DBW 104;
      +I;
      T     DB6.DBW 104;
M037: NOP   0;
      A     L 0.0;
      A(;
      L     DB6.DBW 104;
      L     1;
      >=I;
      );
      =     DB6.DBX 98.0;
NETWORK
TITLE =
      A     DB6.DBX 98.0;
      A     DB6.DBX 0.2;
      =     L 0.0;
      A     L 0.0;
      AN    DB6.DBX 106.1;
      A     M 0.3;
      JNB   M038;
      L     1;
      L     DB6.DBW 110;
      +I;
      T     DB6.DBW 110;
M038: NOP   0;
      A     L 0.0;
      A(;
      L     DB6.DBW 110;
      L     DB6.DBW 108;
      >=I;
      );
      =     DB6.DBX 106.1;
NETWORK
TITLE =
      A     M 0.1;
      A(;
      A     DB6.DBX 7.5;
      A     M 0.2;
      O     DB6.DBX 98.0;
      O     DB1.DBX 0.5;
      );
      =     DB6.DBX 280.1;
